  STRUCT
   HLINE_DX : STRUCT
    REP_SEL : BOOL ;
    S02_SEL : BOOL ;
    S03_SEL : BOOL ;
    RC2_SEL : BOOL ;
    BUF2_SEL : BOOL ;
    S04_SEL : BOOL ;
    S05_SEL : BOOL ;
    TT_SEL : BOOL ;
    SPARE : BOOL ;
    SPARE1 : BOOL ;
    SPARE2 : BOOL ;
    SPARE3 : BOOL ;
    SPARE4 : BOOL ;
    SPARE5 : BOOL ;
    SPARE6 : BOOL ;
    SPARE7 : BOOL ;
    SPARE8 : BOOL ;
    SPARE9 : BOOL ;
    SPARE10 : BOOL ;
    SPARE11 : BOOL ;
    SPARE12 : BOOL ;
    SPARE13 : BOOL ;
    SPARE14 : BOOL ;
    SPARE15 : BOOL ;
    SPARE16 : BOOL ;
    SPARE17 : BOOL ;
    SPARE18 : BOOL ;
    SPARE19 : BOOL ;
    SPARE20 : BOOL ;
    SPARE21 : BOOL ;
    PB_ADV : BOOL ;
    PB_RET : BOOL ;
    LCK1_SEL : BOOL ;
    STP1_SEL : BOOL ;
    LCK2_SEL : BOOL ;
    STP2_SEL : BOOL ;
    LCK3_SEL : BOOL ;
    STP3_SEL : BOOL ;
    LCK4_SEL : BOOL ;
    STP4_SEL : BOOL ;
    ELE_SEL : BOOL ;
    RC_SEL : BOOL ;
    HK_SEL : BOOL ;
    PLOCK_SEL : BOOL ;
    MOTOR_SEL : BOOL ;
    SPARE37 : BOOL ;
    SPARE38 : BOOL ;
    SPARE39 : BOOL ;
    SPARE40 : BOOL ;
    SPARE41 : BOOL ;
    SPARE42 : BOOL ;
    SPARE43 : BOOL ;
    SPARE44 : BOOL ;
    SPARE45 : BOOL ;
    SPARE46 : BOOL ;
    SPARE47 : BOOL ;
    SPARE48 : BOOL ;
    SPARE49 : BOOL ;
    SPARE50 : BOOL ;
    SPARE51 : BOOL ;
    SPARE52 : BOOL ;
    SPARE53 : BOOL ;
    SPARE54 : BOOL ;
    SPARE55 : BOOL ;
    REP_LCK1_SEL : BOOL ;
    REP_STP1_SEL : BOOL ;
    REP_LCK2_SEL : BOOL ;
    REP_STP2_SEL : BOOL ;
    SPARE60 : BOOL ;
    SPARE61 : BOOL ;
    SPARE62 : BOOL ;
    SPARE63 : BOOL ;
    REP_ELE_SEL : BOOL ;
    REP_RC_SEL : BOOL ;
    SPARE66 : BOOL ;
    SPARE67 : BOOL ;
    SPARE68 : BOOL ;
    SPARE69 : BOOL ;
    SPARE70 : BOOL ;
    SPARE71 : BOOL ;
    S02_LCK1_SEL : BOOL ;
    S02_STP1_SEL : BOOL ;
    S02_LCK2_SEL : BOOL ;
    S02_STP2_SEL : BOOL ;
    S02_LCK3_SEL : BOOL ;
    S02_STP3_SEL : BOOL ;
    SPARE78 : BOOL ;
    SPARE79 : BOOL ;
    S02_ELE_SEL : BOOL ;
    S02_RC_SEL : BOOL ;
    SPARE22 : BOOL ;
    SPARE23 : BOOL ;
    SPARE84 : BOOL ;
    SPARE85 : BOOL ;
    SPARE86 : BOOL ;
    SPARE87 : BOOL ;
    S03_LCK1_SEL : BOOL ;
    S03_STP1_SEL : BOOL ;
    SPARE90 : BOOL ;
    SPARE91 : BOOL ;
    SPARE92 : BOOL ;
    SPARE93 : BOOL ;
    SPARE94 : BOOL ;
    SPARE95 : BOOL ;
    S03_ELE_SEL : BOOL ;
    SPARE97 : BOOL ;
    SPARE98 : BOOL ;
    SPARE99 : BOOL ;
    SPARE100 : BOOL ;
    SPARE101 : BOOL ;
    SPARE102 : BOOL ;
    SPARE103 : BOOL ;
    RC2_LCK1_SEL : BOOL ;
    RC2_STP1_SEL : BOOL ;
    RC2_LCK2_SEL : BOOL ;
    RC2_STP2_SEL : BOOL ;
    RC2_LCK3_SEL : BOOL ;
    RC2_STP3_SEL : BOOL ;
    RC2_LCK4_SEL : BOOL ;
    RC2_STP4_SEL : BOOL ;
    SPARE112 : BOOL ;
    RC2_RC_SEL : BOOL ;
    SPARE114 : BOOL ;
    SPARE115 : BOOL ;
    SPARE116 : BOOL ;
    SPARE117 : BOOL ;
    SPARE118 : BOOL ;
    SPARE119 : BOOL ;
    BUF1_LCK1_SEL : BOOL ;
    BUF1_STP1_SEL : BOOL ;
    SPARE122 : BOOL ;
    SPARE123 : BOOL ;
    SPARE124 : BOOL ;
    SPARE125 : BOOL ;
    SPARE126 : BOOL ;
    SPARE127 : BOOL ;
    SPARE128 : BOOL ;
    SPARE129 : BOOL ;
    SPARE130 : BOOL ;
    SPARE131 : BOOL ;
    SPARE132 : BOOL ;
    SPARE133 : BOOL ;
    SPARE134 : BOOL ;
    SPARE135 : BOOL ;
    BUF2_LCK1_SEL : BOOL ;
    BUF2_STP1_SEL : BOOL ;
    SPARE138 : BOOL ;
    SPARE139 : BOOL ;
    SPARE140 : BOOL ;
    SPARE141 : BOOL ;
    SPARE142 : BOOL ;
    SPARE143 : BOOL ;
    SPARE144 : BOOL ;
    SPARE145 : BOOL ;
    SPARE146 : BOOL ;
    SPARE147 : BOOL ;
    SPARE148 : BOOL ;
    SPARE149 : BOOL ;
    SPARE150 : BOOL ;
    SPARE151 : BOOL ;
    S04_LCK1_SEL : BOOL ;
    S04_STP1_SEL : BOOL ;
    SPARE154 : BOOL ;
    SPARE155 : BOOL ;
    SPARE156 : BOOL ;
    SPARE157 : BOOL ;
    SPARE158 : BOOL ;
    SPARE159 : BOOL ;
    S04_ELE_SEL : BOOL ;
    SPARE161 : BOOL ;
    S04_HK_SEL : BOOL ;
    SPARE163 : BOOL ;
    SPARE164 : BOOL ;
    SPARE165 : BOOL ;
    SPARE166 : BOOL ;
    SPARE167 : BOOL ;
    S05_LCK1_SEL : BOOL ;
    S05_STP1_SEL : BOOL ;
    SPARE170 : BOOL ;
    SPARE171 : BOOL ;
    SPARE172 : BOOL ;
    SPARE173 : BOOL ;
    SPARE174 : BOOL ;
    SPARE175 : BOOL ;
    S05_ELE_SEL : BOOL ;
    SPARE177 : BOOL ;
    S05_HK_SEL : BOOL ;
    SPARE179 : BOOL ;
    SPARE180 : BOOL ;
    SPARE181 : BOOL ;
    SPARE182 : BOOL ;
    SPARE183 : BOOL ;
    TT_PLOCK_SEL : BOOL ;
    TT_ELE_SEL : BOOL ;
    TT_ROLL_SEL : BOOL ;
    SPARE187 : BOOL ;
    SPARE188 : BOOL ;
    SPARE189 : BOOL ;
    SPARE190 : BOOL ;
    SPARE191 : BOOL ;
    SPARE192 : BOOL ;
    SPARE193 : BOOL ;
    SPARE194 : BOOL ;
    SPARE195 : BOOL ;
    SPARE196 : BOOL ;
    SPARE197 : BOOL ;
    SPARE198 : BOOL ;
    SPARE199 : BOOL ;
    SPARE200 : BOOL ;
    SPARE201 : BOOL ;
    SPARE202 : BOOL ;
    SPARE203 : BOOL ;
    SPARE204 : BOOL ;
    SPARE205 : BOOL ;
    SPARE206 : BOOL ;
    SPARE207 : BOOL ;
    SPARE208 : BOOL ;
    SPARE209 : BOOL ;
    SPARE210 : BOOL ;
    SPARE211 : BOOL ;
    SPARE212 : BOOL ;
    SPARE213 : BOOL ;
    SPARE214 : BOOL ;
    SPARE215 : BOOL ;
    SPARE216 : BOOL ;
    SPARE217 : BOOL ;
    SPARE218 : BOOL ;
    SPARE219 : BOOL ;
    SPARE220 : BOOL ;
    SPARE221 : BOOL ;
    SPARE222 : BOOL ;
    SPARE223 : BOOL ;
    SPARE224 : BOOL ;
    SPARE225 : BOOL ;
    SPARE226 : BOOL ;
    SPARE227 : BOOL ;
    SPARE228 : BOOL ;
    SPARE229 : BOOL ;
    SPARE230 : BOOL ;
    SPARE231 : BOOL ;
    SPARE232 : BOOL ;
    SPARE233 : BOOL ;
    SPARE234 : BOOL ;
    SPARE235 : BOOL ;
    SPARE236 : BOOL ;
    SPARE237 : BOOL ;
    SPARE238 : BOOL ;
    SPARE239 : BOOL ;
    SPARE240 : BOOL ;
    SPARE241 : BOOL ;
    SPARE242 : BOOL ;
    SPARE243 : BOOL ;
    SPARE244 : BOOL ;
    SPARE245 : BOOL ;
    SPARE246 : BOOL ;
    SPARE247 : BOOL ;
    SPARE248 : BOOL ;
    SPARE249 : BOOL ;
    SPARE250 : BOOL ;
    SPARE251 : BOOL ;
    SPARE252 : BOOL ;
    SPARE253 : BOOL ;
    SPARE254 : BOOL ;
    SPARE255 : BOOL ;
    SPARE256 : BOOL ;
    SPARE257 : BOOL ;
    SPARE258 : BOOL ;
    SPARE259 : BOOL ;
    SPARE260 : BOOL ;
    SPARE261 : BOOL ;
    SPARE262 : BOOL ;
    SPARE263 : BOOL ;
    SPARE264 : BOOL ;
    SPARE265 : BOOL ;
    SPARE266 : BOOL ;
    SPARE267 : BOOL ;
    SPARE268 : BOOL ;
    SPARE269 : BOOL ;
    SPARE270 : BOOL ;
    SPARE271 : BOOL ;
    SPARE272 : BOOL ;
    SPARE273 : BOOL ;
    SPARE274 : BOOL ;
    SPARE275 : BOOL ;
    SPARE276 : BOOL ;
    SPARE277 : BOOL ;
    SPARE278 : BOOL ;
    SPARE279 : BOOL ;
    SPARE280 : BOOL ;
    SPARE281 : BOOL ;
    SPARE282 : BOOL ;
    SPARE283 : BOOL ;
    SPARE284 : BOOL ;
    SPARE285 : BOOL ;
    SPARE286 : BOOL ;
    SPARE287 : BOOL ;
    SPARE288 : BOOL ;
    SPARE289 : BOOL ;
    SPARE290 : BOOL ;
    SPARE291 : BOOL ;
    SPARE292 : BOOL ;
    SPARE293 : BOOL ;
    SPARE294 : BOOL ;
    SPARE295 : BOOL ;
    SPARE296 : BOOL ;
    SPARE297 : BOOL ;
    SPARE298 : BOOL ;
    SPARE299 : BOOL ;
    SPARE300 : BOOL ;
    SPARE301 : BOOL ;
    SPARE302 : BOOL ;
    SPARE303 : BOOL ;
    SPARE304 : BOOL ;
    SPARE305 : BOOL ;
    SPARE306 : BOOL ;
    SPARE307 : BOOL ;
    SPARE308 : BOOL ;
    SPARE309 : BOOL ;
    SPARE310 : BOOL ;
   END_STRUCT ;
   HLINE_DW : STRUCT
    REP_LCK1_A_LAMP : WORD ;
    REP_LCK1_R_LAMP : WORD ;
    REP_STP1_A_LAMP : WORD ;
    REP_STP1_R_LAMP : WORD ;
    REP_LCK2_A_LAMP : WORD ;
    REP_LCK2_R_LAMP : WORD ;
    REP_STP2_A_LAMP : WORD ;
    REP_STP2_R_LAMP : WORD ;
    REP_ELE_A_LAMP : WORD ;
    REP_ELE_R_LAMP : WORD ;
    REP_RC_A_LAMP : WORD ;
    REP_RC_R_LAMP : WORD ;
    SPARE_WORD1 : WORD ;
    SPARE_WORD2 : WORD ;
    SPARE_WORD3 : WORD ;
    SPARE_WORD4 : WORD ;
    S02_LCK1_A_LAMP : WORD ;
    S02_LCK1_R_LAMP : WORD ;
    S02_STP1_A_LAMP : WORD ;
    S02_STP1_R_LAMP : WORD ;
    S02_LCK2_A_LAMP : WORD ;
    S02_LCK2_R_LAMP : WORD ;
    S02_STP2_A_LAMP : WORD ;
    S02_STP2_R_LAMP : WORD ;
    S02_LCK3_A_LAMP : WORD ;
    S02_LCK3_R_LAMP : WORD ;
    S02_STP3_A_LAMP : WORD ;
    S02_STP3_R_LAMP : WORD ;
    S02_ELE_A_LAMP : WORD ;
    S02_ELE_R_LAMP : WORD ;
    S02_RC_A_LAMP : WORD ;
    S02_RC_R_LAMP : WORD ;
    SPARE_WORD15 : WORD ;
    SPARE_WORD16 : WORD ;
    SPARE_WORD17 : WORD ;
    SPARE_WORD18 : WORD ;
    S03_LCK1_A_LAMP : WORD ;
    S03_LCK1_R_LAMP : WORD ;
    S03_STP1_A_LAMP : WORD ;
    S03_STP1_R_LAMP : WORD ;
    S03_ELE_A_LAMP : WORD ;
    S03_ELE_R_LAMP : WORD ;
    SPARE_WORD25 : WORD ;
    SPARE_WORD26 : WORD ;
    SPARE_WORD27 : WORD ;
    SPARE_WORD28 : WORD ;
    RC2_LCK1_A_LAMP : WORD ;
    RC2_LCK1_R_LAMP : WORD ;
    RC2_STP1_A_LAMP : WORD ;
    RC2_STP1_R_LAMP : WORD ;
    RC2_LCK2_A_LAMP : WORD ;
    RC2_LCK2_R_LAMP : WORD ;
    RC2_STP2_A_LAMP : WORD ;
    RC2_STP2_R_LAMP : WORD ;
    RC2_LCK3_A_LAMP1 : WORD ;
    RC2_LCK3_R_LAMP1 : WORD ;
    RC2_STP3_A_LAMP1 : WORD ;
    RC2_STP3_R_LAMP1 : WORD ;
    RC2_LCK4_A_LAMP1 : WORD ;
    RC2_LCK4_R_LAMP1 : WORD ;
    RC2_STP4_A_LAMP1 : WORD ;
    RC2_STP4_R_LAMP1 : WORD ;
    RC2_RC_A_LAMP1 : WORD ;
    RC2_RC_R_LAMP1 : WORD ;
    SPARE_WORD34 : WORD ;
    SPARE_WORD35 : WORD ;
    SPARE_WORD36 : WORD ;
    SPARE_WORD37 : WORD ;
    BUF1_LCK1_A_LAMP : WORD ;
    BUF1_LCK1_R_LAMP : WORD ;
    BUF1_STP1_A_LAMP : WORD ;
    BUF1_STP1_R_LAMP : WORD ;
    SPARE_WORD42 : WORD ;
    SPARE_WORD43 : WORD ;
    SPARE_WORD44 : WORD ;
    SPARE_WORD45 : WORD ;
    BUF2_LCK1_A_LAMP : WORD ;
    BUF2_LCK1_R_LAMP : WORD ;
    BUF2_STP1_A_LAMP : WORD ;
    BUF2_STP1_R_LAMP : WORD ;
    SPARE_WORD50 : WORD ;
    SPARE_WORD51 : WORD ;
    SPARE_WORD52 : WORD ;
    SPARE_WORD53 : WORD ;
    S04_LCK1_A_LAMP : WORD ;
    S04_LCK1_R_LAMP : WORD ;
    S04_STP1_A_LAMP : WORD ;
    S04_STP2_R_LAMP : WORD ;
    S04_ELE_A_LAMP : WORD ;
    S04_ELE_R_LAMP : WORD ;
    S04_HK_A_LAMP : WORD ;
    S04_HK_R_LAMP : WORD ;
    SPARE_WORD55 : WORD ;
    SPARE_WORD56 : WORD ;
    SPARE_WORD57 : WORD ;
    SPARE_WORD58 : WORD ;
    S05_LCK1_A_LAMP : WORD ;
    S05_LCK1_R_LAMP : WORD ;
    S05_STP1_A_LAMP : WORD ;
    S05_STP2_R_LAMP : WORD ;
    S05_ELE_A_LAMP : WORD ;
    S05_ELE_R_LAMP : WORD ;
    S05_HK_A_LAMP : WORD ;
    S05_HK_R_LAMP : WORD ;
    SPARE_WORD60 : WORD ;
    SPARE_WORD61 : WORD ;
    SPARE_WORD62 : WORD ;
    SPARE_WORD63 : WORD ;
    TT_PLOCK_A_LAMP : WORD ;
    TT_PLOCK_R_LAMP : WORD ;
    TT_ELE_A_LAMP : WORD ;
    TT_ELE_R_LAMP : WORD ;
    TT_ROLL_A_LAMP : WORD ;
    TT_ROLL_R_LAMP : WORD ;
    SPARE_WORD70 : WORD ;
    SPARE_WORD71 : WORD ;
    SPARE_WORD72 : WORD ;
    SPARE_WORD73 : WORD ;
    SPARE_WORD74 : WORD ;
    SPARE_WORD75 : WORD ;
    SPARE_WORD76 : WORD ;
    SPARE_WORD77 : WORD ;
    SPARE_WORD78 : WORD ;
    SPARE_WORD79 : WORD ;
    SPARE_WORD80 : WORD ;
    SPARE_WORD81 : WORD ;
    SPARE_WORD82 : WORD ;
    SPARE_WORD83 : WORD ;
    SPARE_WORD84 : WORD ;
    SPARE_WORD85 : WORD ;
    SPARE_WORD86 : WORD ;
    SPARE_WORD87 : WORD ;
    SPARE_WORD88 : WORD ;
    SPARE_WORD89 : WORD ;
    SPARE_WORD90 : WORD ;
    SPARE_WORD91 : WORD ;
    SPARE_WORD92 : WORD ;
    SPARE_WORD93 : WORD ;
    SPARE_WORD94 : WORD ;
    SPARE_WORD95 : WORD ;
    SPARE_WORD96 : WORD ;
    SPARE_WORD97 : WORD ;
    SPARE_WORD98 : WORD ;
    SPARE_WORD99 : WORD ;
    SPARE_WORD100 : WORD ;
    SPARE_WORD101 : WORD ;
    SPARE_WORD102 : WORD ;
    SPARE_WORD103 : WORD ;
    SPARE_WORD104 : WORD ;
    SPARE_WORD105 : WORD ;
    SPARE_WORD106 : WORD ;
    SPARE_WORD107 : WORD ;
    SPARE_WORD108 : WORD ;
    SPARE_WORD109 : WORD ;
    SPARE_WORD110 : WORD ;
    SPARE_WORD111 : WORD ;
    SPARE_WORD112 : WORD ;
    SPARE_WORD113 : WORD ;
    SPARE_WORD114 : WORD ;
    SPARE_WORD115 : WORD ;
    SPARE_WORD116 : WORD ;
    SPARE_WORD117 : WORD ;
    SPARE_WORD118 : WORD ;
    SPARE_WORD119 : WORD ;
    SPARE_WORD120 : WORD ;
    SPARE_WORD121 : WORD ;
    SPARE_WORD122 : WORD ;
    SPARE_WORD123 : WORD ;
    SPARE_WORD124 : WORD ;
    SPARE_WORD125 : WORD ;
    SPARE_WORD126 : WORD ;
    SPARE_WORD127 : WORD ;
    SPARE_WORD128 : WORD ;
    SPARE_WORD129 : WORD ;
    SPARE_WORD130 : WORD ;
    SPARE_WORD131 : WORD ;
    SPARE_WORD132 : WORD ;
    SPARE_WORD133 : WORD ;
    SPARE_WORD134 : WORD ;
    SPARE_WORD135 : WORD ;
   END_STRUCT ;
   HUPDL_DX : STRUCT
    _1ST_U_SEL : BOOL ;
    _2ND_U1_SEL : BOOL ;
    _2ND_U2_SEL : BOOL ;
    SPUSH1_SEL : BOOL ;
    LOCKG_SEL : BOOL ;
    SPARE1 : BOOL ;
    SPARE2 : BOOL ;
    SPARE3 : BOOL ;
    Q_1ST_PIN_SEL : BOOL ;
    Q_2ND_UNIT_SEL : BOOL ;
    Q_3RD_UNIT_SEL : BOOL ;
    Q_4TH_UNIT_SEL : BOOL ;
    SPARE8 : BOOL ;
    SPARE9 : BOOL ;
    SPARE10 : BOOL ;
    SPARE11 : BOOL ;
    SPARE12 : BOOL ;
    SPARE13 : BOOL ;
    SPARE14 : BOOL ;
    SPARE15 : BOOL ;
    SPARE16 : BOOL ;
    SPARE17 : BOOL ;
    SPARE18 : BOOL ;
    SPARE19 : BOOL ;
    SPARE20 : BOOL ;
    SPARE21 : BOOL ;
    SPARE22 : BOOL ;
    SPARE23 : BOOL ;
    SPARE24 : BOOL ;
    SPARE25 : BOOL ;
    PB_ADV : BOOL ;
    PB_RET : BOOL ;
    BH_1_SEL : BOOL ;
    BH_2_SEL : BOOL ;
    BH_3_SEL : BOOL ;
    BH_4_SEL : BOOL ;
    BH_5_SEL : BOOL ;
    BH_6_SEL : BOOL ;
    BH_7_SEL : BOOL ;
    BH_8_SEL : BOOL ;
    BH_9_SEL : BOOL ;
    BH_10_SEL : BOOL ;
    BH_11_SEL : BOOL ;
    BH_12_SEL : BOOL ;
    BH_13_SEL : BOOL ;
    BH_14_SEL : BOOL ;
    BH_15_SEL : BOOL ;
    BH_16_SEL : BOOL ;
    SPARE42 : BOOL ;
    SPARE43 : BOOL ;
    SPARE44 : BOOL ;
    SPARE45 : BOOL ;
    SPARE46 : BOOL ;
    SPARE47 : BOOL ;
    SPARE48 : BOOL ;
    SPARE49 : BOOL ;
    SPARE50 : BOOL ;
    SPARE51 : BOOL ;
    SPARE52 : BOOL ;
    SPARE53 : BOOL ;
    SPARE54 : BOOL ;
    SPARE55 : BOOL ;
    SPARE56 : BOOL ;
    SPARE57 : BOOL ;
    VI_1_SEL : BOOL ;
    VI_2_SEL : BOOL ;
    VI_3_SEL : BOOL ;
    VI_4_SEL : BOOL ;
    VI_5_SEL : BOOL ;
    VI_6_SEL : BOOL ;
    VI_7_SEL : BOOL ;
    VI_8_SEL : BOOL ;
    VI_9_SEL : BOOL ;
    VI_10_SEL : BOOL ;
    VI_11_SEL : BOOL ;
    VI_12_SEL : BOOL ;
    VI_13_SEL : BOOL ;
    VI_14_SEL : BOOL ;
    VI_15_SEL : BOOL ;
    VI_16_SEL : BOOL ;
    SPARE59 : BOOL ;
    SPARE60 : BOOL ;
    SPARE61 : BOOL ;
    SPARE62 : BOOL ;
    SPARE63 : BOOL ;
    SPARE64 : BOOL ;
    SPARE65 : BOOL ;
    SPARE66 : BOOL ;
    SPARE67 : BOOL ;
    SPARE68 : BOOL ;
    SPARE69 : BOOL ;
    SPARE70 : BOOL ;
    SPARE71 : BOOL ;
    SPARE72 : BOOL ;
    SPARE73 : BOOL ;
    SPARE74 : BOOL ;
    SPARE75 : BOOL ;
    SPARE76 : BOOL ;
    SPARE77 : BOOL ;
    SPARE78 : BOOL ;
    SPARE79 : BOOL ;
    SPARE80 : BOOL ;
    SPARE81 : BOOL ;
    SPARE82 : BOOL ;
    SPARE83 : BOOL ;
    SPARE84 : BOOL ;
    SPARE85 : BOOL ;
    SPARE86 : BOOL ;
    SPARE87 : BOOL ;
    SPARE88 : BOOL ;
    SPARE89 : BOOL ;
    SPARE90 : BOOL ;
    SPARE91 : BOOL ;
    SPARE92 : BOOL ;
    SPARE93 : BOOL ;
    SPARE94 : BOOL ;
    SPARE95 : BOOL ;
    SPARE96 : BOOL ;
    SPARE97 : BOOL ;
    SPARE98 : BOOL ;
    SPARE99 : BOOL ;
    SPARE100 : BOOL ;
    SPARE101 : BOOL ;
    SPARE102 : BOOL ;
    SPARE103 : BOOL ;
    SPARE104 : BOOL ;
    SPARE105 : BOOL ;
    SPARE106 : BOOL ;
    SPARE107 : BOOL ;
    SPARE108 : BOOL ;
    SPARE109 : BOOL ;
    SPARE110 : BOOL ;
    SPARE111 : BOOL ;
    SPARE112 : BOOL ;
    SPARE113 : BOOL ;
    SPARE114 : BOOL ;
    SPARE115 : BOOL ;
    SPARE116 : BOOL ;
    SPARE117 : BOOL ;
    SPARE118 : BOOL ;
    SPARE119 : BOOL ;
    SPARE120 : BOOL ;
    SPARE121 : BOOL ;
    SPARE122 : BOOL ;
    SPARE123 : BOOL ;
    SPARE124 : BOOL ;
    SPARE125 : BOOL ;
    SPARE126 : BOOL ;
    SPARE127 : BOOL ;
    SPARE128 : BOOL ;
    SPARE129 : BOOL ;
    SPARE130 : BOOL ;
    SPARE131 : BOOL ;
    SPARE132 : BOOL ;
    SPARE133 : BOOL ;
    SPARE134 : BOOL ;
    SPARE135 : BOOL ;
    SPARE136 : BOOL ;
    SPARE137 : BOOL ;
    SPARE138 : BOOL ;
   END_STRUCT ;
   HUPDL_DW : STRUCT
    _1ST_U_ADV_LAMP : WORD ;
    _1ST_U_RET_LAMP : WORD ;
    _2ND_U1_ADV_LAMP : WORD ;
    _2ND_U1_RET_LAMP : WORD ;
    _2ND_U2_ADV_LAMP : WORD ;
    _2ND_U2_RET_LAMP : WORD ;
    SPUSH1_ADV_LAMP : WORD ;
    SPUSH1_RET_LAMP : WORD ;
    LOCKG_ADV_LAMP : WORD ;
    LOCKG_RET_LAMP : WORD ;
    SPARE_WORD2 : WORD ;
    SPARE_WORD3 : WORD ;
    SPARE_WORD4 : WORD ;
    SPARE_WORD5 : WORD ;
    SPARE_WORD6 : WORD ;
    SPARE_WORD7 : WORD ;
    SPARE_WORD8 : WORD ;
    SPARE_WORD9 : WORD ;
    SPARE_WORD10 : WORD ;
    SPARE_WORD11 : WORD ;
    Q_1ST_PIN_ADV_LAMP : WORD ;
    Q_1ST_PIN_RET_LAMP : WORD ;
    Q_2ND_UNIT_ADV_LAMP : WORD ;
    Q_2ND_UNIT_RET_LAMP : WORD ;
    Q_3RD_UNIT_ADV_LAMP : WORD ;
    Q_3RD_UNIT_RET_LAMP : WORD ;
    Q_4TH_UNIT_ADV_LAMP : WORD ;
    Q_4TH_UNIT_RET_LAMP : WORD ;
    SPARE_WORD20 : WORD ;
    SPARE_WORD21 : WORD ;
    SPARE_WORD22 : WORD ;
    SPARE_WORD23 : WORD ;
    BH_1_ADV_LAMP : WORD ;
    BH_1_RET_LAMP : WORD ;
    BH_2_ADV_LAMP : WORD ;
    BH_2_RET_LAMP : WORD ;
    BH_3_ADV_LAMP : WORD ;
    BH_3_RET_LAMP : WORD ;
    BH_4_ADV_LAMP : WORD ;
    BH_4_RET_LAMP : WORD ;
    BH_5_ADV_LAMP : WORD ;
    BH_5_RET_LAMP : WORD ;
    BH_6_ADV_LAMP : WORD ;
    BH_6_RET_LAMP : WORD ;
    BH_7_ADV_LAMP : WORD ;
    BH_7_RET_LAMP : WORD ;
    BH_8_ADV_LAMP : WORD ;
    BH_8_RET_LAMP : WORD ;
    BH_9_ADV_LAMP : WORD ;
    BH_9_RET_LAMP : WORD ;
    BH_10_ADV_LAMP : WORD ;
    BH_10_RET_LAMP : WORD ;
    SPARE_WORD54 : WORD ;
    SPARE_WORD55 : WORD ;
    SPARE_WORD56 : WORD ;
    SPARE_WORD57 : WORD ;
    SPARE_WORD58 : WORD ;
    SPARE_WORD59 : WORD ;
    SPARE_WORD60 : WORD ;
    SPARE_WORD61 : WORD ;
    SPARE_WORD62 : WORD ;
    SPARE_WORD63 : WORD ;
    SPARE_WORD64 : WORD ;
    SPARE_WORD65 : WORD ;
    SPARE_WORD66 : WORD ;
    SPARE_WORD67 : WORD ;
    SPARE_WORD68 : WORD ;
    SPARE_WORD69 : WORD ;
    SPARE_WORD70 : WORD ;
    SPARE_WORD71 : WORD ;
    SPARE_WORD72 : WORD ;
    SPARE_WORD73 : WORD ;
    SPARE_WORD74 : WORD ;
    SPARE_WORD75 : WORD ;
    SPARE_WORD76 : WORD ;
    SPARE_WORD77 : WORD ;
    SPARE_WORD78 : WORD ;
    SPARE_WORD79 : WORD ;
    SPARE_WORD80 : WORD ;
    SPARE_WORD81 : WORD ;
    SPARE_WORD82 : WORD ;
    SPARE_WORD83 : WORD ;
    SPARE_WORD84 : WORD ;
    SPARE_WORD85 : WORD ;
    SPARE_WORD86 : WORD ;
    SPARE_WORD87 : WORD ;
    SPARE_WORD88 : WORD ;
    SPARE_WORD89 : WORD ;
    SPARE_WORD90 : WORD ;
    SPARE_WORD91 : WORD ;
    SPARE_WORD92 : WORD ;
    SPARE_WORD93 : WORD ;
    SPARE_WORD94 : WORD ;
    SPARE_WORD95 : WORD ;
    SPARE_WORD96 : WORD ;
    SPARE_WORD97 : WORD ;
    SPARE_WORD98 : WORD ;
    SPARE_WORD99 : WORD ;
    SPARE_WORD100 : WORD ;
    SPARE_WORD101 : WORD ;
    SPARE_WORD102 : WORD ;
    SPARE_WORD103 : WORD ;
    SPARE_WORD104 : WORD ;
    SPARE_WORD105 : WORD ;
    SPARE_WORD106 : WORD ;
    SPARE_WORD107 : WORD ;
    SPARE_WORD108 : WORD ;
    SPARE_WORD109 : WORD ;
    SPARE_WORD110 : WORD ;
    SPARE_WORD111 : WORD ;
    SPARE_WORD112 : WORD ;
    SPARE_WORD113 : WORD ;
    SPARE_WORD114 : WORD ;
    SPARE_WORD115 : WORD ;
    SPARE_WORD116 : WORD ;
    SPARE_WORD117 : WORD ;
    SPARE_WORD118 : WORD ;
    SPARE_WORD119 : WORD ;
    SPARE_WORD120 : WORD ;
    SPARE_WORD121 : WORD ;
    SPARE_WORD122 : WORD ;
    SPARE_WORD123 : WORD ;
    SPARE_WORD124 : WORD ;
    SPARE_WORD125 : WORD ;
    SPARE_WORD126 : WORD ;
    SPARE_WORD127 : WORD ;
    SPARE_WORD128 : WORD ;
    SPARE_WORD129 : WORD ;
    SPARE_WORD130 : WORD ;
    SPARE_WORD131 : WORD ;
    SPARE_WORD132 : WORD ;
    SPARE_WORD133 : WORD ;
    SPARE_WORD134 : WORD ;
    SPARE_WORD135 : WORD ;
    SPARE_WORD136 : WORD ;
    SPARE_WORD137 : WORD ;
    SPARE_WORD138 : WORD ;
    SPARE_WORD139 : WORD ;
    SPARE_WORD140 : WORD ;
    SPARE_WORD141 : WORD ;
    SPARE_WORD142 : WORD ;
    SPARE_WORD143 : WORD ;
    SPARE_WORD144 : WORD ;
    SPARE_WORD145 : WORD ;
    SPARE_WORD146 : WORD ;
    SPARE_WORD147 : WORD ;
    SPARE_WORD148 : WORD ;
    SPARE_WORD149 : WORD ;
    SPARE_WORD150 : WORD ;
    SPARE_WORD151 : WORD ;
    SPARE_WORD152 : WORD ;
    SPARE_WORD153 : WORD ;
    SPARE_WORD154 : WORD ;
    SPARE_WORD155 : WORD ;
    SPARE_WORD156 : WORD ;
    SPARE_WORD157 : WORD ;
    SPARE_WORD158 : WORD ;
    SPARE_WORD159 : WORD ;
    SPARE_WORD160 : WORD ;
    SPARE_WORD161 : WORD ;
    SPARE_WORD162 : WORD ;
    SPARE_WORD163 : WORD ;
    SPARE_WORD164 : WORD ;
    SPARE_WORD165 : WORD ;
    SPARE_WORD166 : WORD ;
    SPARE_WORD167 : WORD ;
    SPARE_WORD168 : WORD ;
    SPARE_WORD169 : WORD ;
    SPARE_WORD170 : WORD ;
    SPARE_WORD171 : WORD ;
    SPARE_WORD172 : WORD ;
    SPARE_WORD173 : WORD ;
    SPARE_WORD174 : WORD ;
    SPARE_WORD175 : WORD ;
    SPARE_WORD176 : WORD ;
    SPARE_WORD177 : WORD ;
    SPARE_WORD178 : WORD ;
    SPARE_WORD179 : WORD ;
    SPARE_WORD180 : WORD ;
    SPARE_WORD181 : WORD ;
   END_STRUCT ;
  END_STRUCT ;
BEGIN
   HLINE_DX.REP_SEL := FALSE;
   HLINE_DX.S02_SEL := FALSE;
   HLINE_DX.S03_SEL := FALSE;
   HLINE_DX.RC2_SEL := FALSE;
   HLINE_DX.BUF2_SEL := FALSE;
   HLINE_DX.S04_SEL := FALSE;
   HLINE_DX.S05_SEL := FALSE;
   HLINE_DX.TT_SEL := FALSE;
   HLINE_DX.SPARE := FALSE;
   HLINE_DX.SPARE1 := FALSE;
   HLINE_DX.SPARE2 := FALSE;
   HLINE_DX.SPARE3 := FALSE;
   HLINE_DX.SPARE4 := FALSE;
   HLINE_DX.SPARE5 := FALSE;
   HLINE_DX.SPARE6 := FALSE;
   HLINE_DX.SPARE7 := FALSE;
   HLINE_DX.SPARE8 := FALSE;
   HLINE_DX.SPARE9 := FALSE;
   HLINE_DX.SPARE10 := FALSE;
   HLINE_DX.SPARE11 := FALSE;
   HLINE_DX.SPARE12 := FALSE;
   HLINE_DX.SPARE13 := FALSE;
   HLINE_DX.SPARE14 := FALSE;
   HLINE_DX.SPARE15 := FALSE;
   HLINE_DX.SPARE16 := FALSE;
   HLINE_DX.SPARE17 := FALSE;
   HLINE_DX.SPARE18 := FALSE;
   HLINE_DX.SPARE19 := FALSE;
   HLINE_DX.SPARE20 := FALSE;
   HLINE_DX.SPARE21 := FALSE;
   HLINE_DX.PB_ADV := FALSE;
   HLINE_DX.PB_RET := FALSE;
   HLINE_DX.LCK1_SEL := FALSE;
   HLINE_DX.STP1_SEL := FALSE;
   HLINE_DX.LCK2_SEL := FALSE;
   HLINE_DX.STP2_SEL := FALSE;
   HLINE_DX.LCK3_SEL := FALSE;
   HLINE_DX.STP3_SEL := FALSE;
   HLINE_DX.LCK4_SEL := FALSE;
   HLINE_DX.STP4_SEL := FALSE;
   HLINE_DX.ELE_SEL := FALSE;
   HLINE_DX.RC_SEL := FALSE;
   HLINE_DX.HK_SEL := FALSE;
   HLINE_DX.PLOCK_SEL := FALSE;
   HLINE_DX.MOTOR_SEL := FALSE;
   HLINE_DX.SPARE37 := FALSE;
   HLINE_DX.SPARE38 := FALSE;
   HLINE_DX.SPARE39 := FALSE;
   HLINE_DX.SPARE40 := FALSE;
   HLINE_DX.SPARE41 := FALSE;
   HLINE_DX.SPARE42 := FALSE;
   HLINE_DX.SPARE43 := FALSE;
   HLINE_DX.SPARE44 := FALSE;
   HLINE_DX.SPARE45 := FALSE;
   HLINE_DX.SPARE46 := FALSE;
   HLINE_DX.SPARE47 := FALSE;
   HLINE_DX.SPARE48 := FALSE;
   HLINE_DX.SPARE49 := FALSE;
   HLINE_DX.SPARE50 := FALSE;
   HLINE_DX.SPARE51 := FALSE;
   HLINE_DX.SPARE52 := FALSE;
   HLINE_DX.SPARE53 := FALSE;
   HLINE_DX.SPARE54 := FALSE;
   HLINE_DX.SPARE55 := FALSE;
   HLINE_DX.REP_LCK1_SEL := FALSE;
   HLINE_DX.REP_STP1_SEL := FALSE;
   HLINE_DX.REP_LCK2_SEL := FALSE;
   HLINE_DX.REP_STP2_SEL := FALSE;
   HLINE_DX.SPARE60 := FALSE;
   HLINE_DX.SPARE61 := FALSE;
   HLINE_DX.SPARE62 := FALSE;
   HLINE_DX.SPARE63 := FALSE;
   HLINE_DX.REP_ELE_SEL := FALSE;
   HLINE_DX.REP_RC_SEL := FALSE;
   HLINE_DX.SPARE66 := FALSE;
   HLINE_DX.SPARE67 := FALSE;
   HLINE_DX.SPARE68 := FALSE;
   HLINE_DX.SPARE69 := FALSE;
   HLINE_DX.SPARE70 := FALSE;
   HLINE_DX.SPARE71 := FALSE;
   HLINE_DX.S02_LCK1_SEL := FALSE;
   HLINE_DX.S02_STP1_SEL := FALSE;
   HLINE_DX.S02_LCK2_SEL := FALSE;
   HLINE_DX.S02_STP2_SEL := FALSE;
   HLINE_DX.S02_LCK3_SEL := FALSE;
   HLINE_DX.S02_STP3_SEL := FALSE;
   HLINE_DX.SPARE78 := FALSE;
   HLINE_DX.SPARE79 := FALSE;
   HLINE_DX.S02_ELE_SEL := FALSE;
   HLINE_DX.S02_RC_SEL := FALSE;
   HLINE_DX.SPARE22 := FALSE;
   HLINE_DX.SPARE23 := FALSE;
   HLINE_DX.SPARE84 := FALSE;
   HLINE_DX.SPARE85 := FALSE;
   HLINE_DX.SPARE86 := FALSE;
   HLINE_DX.SPARE87 := FALSE;
   HLINE_DX.S03_LCK1_SEL := FALSE;
   HLINE_DX.S03_STP1_SEL := FALSE;
   HLINE_DX.SPARE90 := FALSE;
   HLINE_DX.SPARE91 := FALSE;
   HLINE_DX.SPARE92 := FALSE;
   HLINE_DX.SPARE93 := FALSE;
   HLINE_DX.SPARE94 := FALSE;
   HLINE_DX.SPARE95 := FALSE;
   HLINE_DX.S03_ELE_SEL := FALSE;
   HLINE_DX.SPARE97 := FALSE;
   HLINE_DX.SPARE98 := FALSE;
   HLINE_DX.SPARE99 := FALSE;
   HLINE_DX.SPARE100 := FALSE;
   HLINE_DX.SPARE101 := FALSE;
   HLINE_DX.SPARE102 := FALSE;
   HLINE_DX.SPARE103 := FALSE;
   HLINE_DX.RC2_LCK1_SEL := FALSE;
   HLINE_DX.RC2_STP1_SEL := FALSE;
   HLINE_DX.RC2_LCK2_SEL := FALSE;
   HLINE_DX.RC2_STP2_SEL := FALSE;
   HLINE_DX.RC2_LCK3_SEL := FALSE;
   HLINE_DX.RC2_STP3_SEL := FALSE;
   HLINE_DX.RC2_LCK4_SEL := FALSE;
   HLINE_DX.RC2_STP4_SEL := FALSE;
   HLINE_DX.SPARE112 := FALSE;
   HLINE_DX.RC2_RC_SEL := FALSE;
   HLINE_DX.SPARE114 := FALSE;
   HLINE_DX.SPARE115 := FALSE;
   HLINE_DX.SPARE116 := FALSE;
   HLINE_DX.SPARE117 := FALSE;
   HLINE_DX.SPARE118 := FALSE;
   HLINE_DX.SPARE119 := FALSE;
   HLINE_DX.BUF1_LCK1_SEL := FALSE;
   HLINE_DX.BUF1_STP1_SEL := FALSE;
   HLINE_DX.SPARE122 := FALSE;
   HLINE_DX.SPARE123 := FALSE;
   HLINE_DX.SPARE124 := FALSE;
   HLINE_DX.SPARE125 := FALSE;
   HLINE_DX.SPARE126 := FALSE;
   HLINE_DX.SPARE127 := FALSE;
   HLINE_DX.SPARE128 := FALSE;
   HLINE_DX.SPARE129 := FALSE;
   HLINE_DX.SPARE130 := FALSE;
   HLINE_DX.SPARE131 := FALSE;
   HLINE_DX.SPARE132 := FALSE;
   HLINE_DX.SPARE133 := FALSE;
   HLINE_DX.SPARE134 := FALSE;
   HLINE_DX.SPARE135 := FALSE;
   HLINE_DX.BUF2_LCK1_SEL := FALSE;
   HLINE_DX.BUF2_STP1_SEL := FALSE;
   HLINE_DX.SPARE138 := FALSE;
   HLINE_DX.SPARE139 := FALSE;
   HLINE_DX.SPARE140 := FALSE;
   HLINE_DX.SPARE141 := FALSE;
   HLINE_DX.SPARE142 := FALSE;
   HLINE_DX.SPARE143 := FALSE;
   HLINE_DX.SPARE144 := FALSE;
   HLINE_DX.SPARE145 := FALSE;
   HLINE_DX.SPARE146 := FALSE;
   HLINE_DX.SPARE147 := FALSE;
   HLINE_DX.SPARE148 := FALSE;
   HLINE_DX.SPARE149 := FALSE;
   HLINE_DX.SPARE150 := FALSE;
   HLINE_DX.SPARE151 := FALSE;
   HLINE_DX.S04_LCK1_SEL := FALSE;
   HLINE_DX.S04_STP1_SEL := FALSE;
   HLINE_DX.SPARE154 := FALSE;
   HLINE_DX.SPARE155 := FALSE;
   HLINE_DX.SPARE156 := FALSE;
   HLINE_DX.SPARE157 := FALSE;
   HLINE_DX.SPARE158 := FALSE;
   HLINE_DX.SPARE159 := FALSE;
   HLINE_DX.S04_ELE_SEL := FALSE;
   HLINE_DX.SPARE161 := FALSE;
   HLINE_DX.S04_HK_SEL := FALSE;
   HLINE_DX.SPARE163 := FALSE;
   HLINE_DX.SPARE164 := FALSE;
   HLINE_DX.SPARE165 := FALSE;
   HLINE_DX.SPARE166 := FALSE;
   HLINE_DX.SPARE167 := FALSE;
   HLINE_DX.S05_LCK1_SEL := FALSE;
   HLINE_DX.S05_STP1_SEL := FALSE;
   HLINE_DX.SPARE170 := FALSE;
   HLINE_DX.SPARE171 := FALSE;
   HLINE_DX.SPARE172 := FALSE;
   HLINE_DX.SPARE173 := FALSE;
   HLINE_DX.SPARE174 := FALSE;
   HLINE_DX.SPARE175 := FALSE;
   HLINE_DX.S05_ELE_SEL := FALSE;
   HLINE_DX.SPARE177 := FALSE;
   HLINE_DX.S05_HK_SEL := FALSE;
   HLINE_DX.SPARE179 := FALSE;
   HLINE_DX.SPARE180 := FALSE;
   HLINE_DX.SPARE181 := FALSE;
   HLINE_DX.SPARE182 := FALSE;
   HLINE_DX.SPARE183 := FALSE;
   HLINE_DX.TT_PLOCK_SEL := FALSE;
   HLINE_DX.TT_ELE_SEL := FALSE;
   HLINE_DX.TT_ROLL_SEL := FALSE;
   HLINE_DX.SPARE187 := FALSE;
   HLINE_DX.SPARE188 := FALSE;
   HLINE_DX.SPARE189 := FALSE;
   HLINE_DX.SPARE190 := FALSE;
   HLINE_DX.SPARE191 := FALSE;
   HLINE_DX.SPARE192 := FALSE;
   HLINE_DX.SPARE193 := FALSE;
   HLINE_DX.SPARE194 := FALSE;
   HLINE_DX.SPARE195 := FALSE;
   HLINE_DX.SPARE196 := FALSE;
   HLINE_DX.SPARE197 := FALSE;
   HLINE_DX.SPARE198 := FALSE;
   HLINE_DX.SPARE199 := FALSE;
   HLINE_DX.SPARE200 := FALSE;
   HLINE_DX.SPARE201 := FALSE;
   HLINE_DX.SPARE202 := FALSE;
   HLINE_DX.SPARE203 := FALSE;
   HLINE_DX.SPARE204 := FALSE;
   HLINE_DX.SPARE205 := FALSE;
   HLINE_DX.SPARE206 := FALSE;
   HLINE_DX.SPARE207 := FALSE;
   HLINE_DX.SPARE208 := FALSE;
   HLINE_DX.SPARE209 := FALSE;
   HLINE_DX.SPARE210 := FALSE;
   HLINE_DX.SPARE211 := FALSE;
   HLINE_DX.SPARE212 := FALSE;
   HLINE_DX.SPARE213 := FALSE;
   HLINE_DX.SPARE214 := FALSE;
   HLINE_DX.SPARE215 := FALSE;
   HLINE_DX.SPARE216 := FALSE;
   HLINE_DX.SPARE217 := FALSE;
   HLINE_DX.SPARE218 := FALSE;
   HLINE_DX.SPARE219 := FALSE;
   HLINE_DX.SPARE220 := FALSE;
   HLINE_DX.SPARE221 := FALSE;
   HLINE_DX.SPARE222 := FALSE;
   HLINE_DX.SPARE223 := FALSE;
   HLINE_DX.SPARE224 := FALSE;
   HLINE_DX.SPARE225 := FALSE;
   HLINE_DX.SPARE226 := FALSE;
   HLINE_DX.SPARE227 := FALSE;
   HLINE_DX.SPARE228 := FALSE;
   HLINE_DX.SPARE229 := FALSE;
   HLINE_DX.SPARE230 := FALSE;
   HLINE_DX.SPARE231 := FALSE;
   HLINE_DX.SPARE232 := FALSE;
   HLINE_DX.SPARE233 := FALSE;
   HLINE_DX.SPARE234 := FALSE;
   HLINE_DX.SPARE235 := FALSE;
   HLINE_DX.SPARE236 := FALSE;
   HLINE_DX.SPARE237 := FALSE;
   HLINE_DX.SPARE238 := FALSE;
   HLINE_DX.SPARE239 := FALSE;
   HLINE_DX.SPARE240 := FALSE;
   HLINE_DX.SPARE241 := FALSE;
   HLINE_DX.SPARE242 := FALSE;
   HLINE_DX.SPARE243 := FALSE;
   HLINE_DX.SPARE244 := FALSE;
   HLINE_DX.SPARE245 := FALSE;
   HLINE_DX.SPARE246 := FALSE;
   HLINE_DX.SPARE247 := FALSE;
   HLINE_DX.SPARE248 := FALSE;
   HLINE_DX.SPARE249 := FALSE;
   HLINE_DX.SPARE250 := FALSE;
   HLINE_DX.SPARE251 := FALSE;
   HLINE_DX.SPARE252 := FALSE;
   HLINE_DX.SPARE253 := FALSE;
   HLINE_DX.SPARE254 := FALSE;
   HLINE_DX.SPARE255 := FALSE;
   HLINE_DX.SPARE256 := FALSE;
   HLINE_DX.SPARE257 := FALSE;
   HLINE_DX.SPARE258 := FALSE;
   HLINE_DX.SPARE259 := FALSE;
   HLINE_DX.SPARE260 := FALSE;
   HLINE_DX.SPARE261 := FALSE;
   HLINE_DX.SPARE262 := FALSE;
   HLINE_DX.SPARE263 := FALSE;
   HLINE_DX.SPARE264 := FALSE;
   HLINE_DX.SPARE265 := FALSE;
   HLINE_DX.SPARE266 := FALSE;
   HLINE_DX.SPARE267 := FALSE;
   HLINE_DX.SPARE268 := FALSE;
   HLINE_DX.SPARE269 := FALSE;
   HLINE_DX.SPARE270 := FALSE;
   HLINE_DX.SPARE271 := FALSE;
   HLINE_DX.SPARE272 := FALSE;
   HLINE_DX.SPARE273 := FALSE;
   HLINE_DX.SPARE274 := FALSE;
   HLINE_DX.SPARE275 := FALSE;
   HLINE_DX.SPARE276 := FALSE;
   HLINE_DX.SPARE277 := FALSE;
   HLINE_DX.SPARE278 := FALSE;
   HLINE_DX.SPARE279 := FALSE;
   HLINE_DX.SPARE280 := FALSE;
   HLINE_DX.SPARE281 := FALSE;
   HLINE_DX.SPARE282 := FALSE;
   HLINE_DX.SPARE283 := FALSE;
   HLINE_DX.SPARE284 := FALSE;
   HLINE_DX.SPARE285 := FALSE;
   HLINE_DX.SPARE286 := FALSE;
   HLINE_DX.SPARE287 := FALSE;
   HLINE_DX.SPARE288 := FALSE;
   HLINE_DX.SPARE289 := FALSE;
   HLINE_DX.SPARE290 := FALSE;
   HLINE_DX.SPARE291 := FALSE;
   HLINE_DX.SPARE292 := FALSE;
   HLINE_DX.SPARE293 := FALSE;
   HLINE_DX.SPARE294 := FALSE;
   HLINE_DX.SPARE295 := FALSE;
   HLINE_DX.SPARE296 := FALSE;
   HLINE_DX.SPARE297 := FALSE;
   HLINE_DX.SPARE298 := FALSE;
   HLINE_DX.SPARE299 := FALSE;
   HLINE_DX.SPARE300 := FALSE;
   HLINE_DX.SPARE301 := FALSE;
   HLINE_DX.SPARE302 := FALSE;
   HLINE_DX.SPARE303 := FALSE;
   HLINE_DX.SPARE304 := FALSE;
   HLINE_DX.SPARE305 := FALSE;
   HLINE_DX.SPARE306 := FALSE;
   HLINE_DX.SPARE307 := FALSE;
   HLINE_DX.SPARE308 := FALSE;
   HLINE_DX.SPARE309 := FALSE;
   HLINE_DX.SPARE310 := FALSE;
   HLINE_DW.REP_LCK1_A_LAMP := W#16#0;
   HLINE_DW.REP_LCK1_R_LAMP := W#16#0;
   HLINE_DW.REP_STP1_A_LAMP := W#16#0;
   HLINE_DW.REP_STP1_R_LAMP := W#16#0;
   HLINE_DW.REP_LCK2_A_LAMP := W#16#0;
   HLINE_DW.REP_LCK2_R_LAMP := W#16#0;
   HLINE_DW.REP_STP2_A_LAMP := W#16#0;
   HLINE_DW.REP_STP2_R_LAMP := W#16#0;
   HLINE_DW.REP_ELE_A_LAMP := W#16#0;
   HLINE_DW.REP_ELE_R_LAMP := W#16#0;
   HLINE_DW.REP_RC_A_LAMP := W#16#0;
   HLINE_DW.REP_RC_R_LAMP := W#16#0;
   HLINE_DW.SPARE_WORD1 := W#16#0;
   HLINE_DW.SPARE_WORD2 := W#16#0;
   HLINE_DW.SPARE_WORD3 := W#16#0;
   HLINE_DW.SPARE_WORD4 := W#16#0;
   HLINE_DW.S02_LCK1_A_LAMP := W#16#0;
   HLINE_DW.S02_LCK1_R_LAMP := W#16#0;
   HLINE_DW.S02_STP1_A_LAMP := W#16#0;
   HLINE_DW.S02_STP1_R_LAMP := W#16#0;
   HLINE_DW.S02_LCK2_A_LAMP := W#16#0;
   HLINE_DW.S02_LCK2_R_LAMP := W#16#0;
   HLINE_DW.S02_STP2_A_LAMP := W#16#0;
   HLINE_DW.S02_STP2_R_LAMP := W#16#0;
   HLINE_DW.S02_LCK3_A_LAMP := W#16#0;
   HLINE_DW.S02_LCK3_R_LAMP := W#16#0;
   HLINE_DW.S02_STP3_A_LAMP := W#16#0;
   HLINE_DW.S02_STP3_R_LAMP := W#16#0;
   HLINE_DW.S02_ELE_A_LAMP := W#16#0;
   HLINE_DW.S02_ELE_R_LAMP := W#16#0;
   HLINE_DW.S02_RC_A_LAMP := W#16#0;
   HLINE_DW.S02_RC_R_LAMP := W#16#0;
   HLINE_DW.SPARE_WORD15 := W#16#0;
   HLINE_DW.SPARE_WORD16 := W#16#0;
   HLINE_DW.SPARE_WORD17 := W#16#0;
   HLINE_DW.SPARE_WORD18 := W#16#0;
   HLINE_DW.S03_LCK1_A_LAMP := W#16#0;
   HLINE_DW.S03_LCK1_R_LAMP := W#16#0;
   HLINE_DW.S03_STP1_A_LAMP := W#16#0;
   HLINE_DW.S03_STP1_R_LAMP := W#16#0;
   HLINE_DW.S03_ELE_A_LAMP := W#16#0;
   HLINE_DW.S03_ELE_R_LAMP := W#16#0;
   HLINE_DW.SPARE_WORD25 := W#16#0;
   HLINE_DW.SPARE_WORD26 := W#16#0;
   HLINE_DW.SPARE_WORD27 := W#16#0;
   HLINE_DW.SPARE_WORD28 := W#16#0;
   HLINE_DW.RC2_LCK1_A_LAMP := W#16#0;
   HLINE_DW.RC2_LCK1_R_LAMP := W#16#0;
   HLINE_DW.RC2_STP1_A_LAMP := W#16#0;
   HLINE_DW.RC2_STP1_R_LAMP := W#16#0;
   HLINE_DW.RC2_LCK2_A_LAMP := W#16#0;
   HLINE_DW.RC2_LCK2_R_LAMP := W#16#0;
   HLINE_DW.RC2_STP2_A_LAMP := W#16#0;
   HLINE_DW.RC2_STP2_R_LAMP := W#16#0;
   HLINE_DW.RC2_LCK3_A_LAMP1 := W#16#0;
   HLINE_DW.RC2_LCK3_R_LAMP1 := W#16#0;
   HLINE_DW.RC2_STP3_A_LAMP1 := W#16#0;
   HLINE_DW.RC2_STP3_R_LAMP1 := W#16#0;
   HLINE_DW.RC2_LCK4_A_LAMP1 := W#16#0;
   HLINE_DW.RC2_LCK4_R_LAMP1 := W#16#0;
   HLINE_DW.RC2_STP4_A_LAMP1 := W#16#0;
   HLINE_DW.RC2_STP4_R_LAMP1 := W#16#0;
   HLINE_DW.RC2_RC_A_LAMP1 := W#16#0;
   HLINE_DW.RC2_RC_R_LAMP1 := W#16#0;
   HLINE_DW.SPARE_WORD34 := W#16#0;
   HLINE_DW.SPARE_WORD35 := W#16#0;
   HLINE_DW.SPARE_WORD36 := W#16#0;
   HLINE_DW.SPARE_WORD37 := W#16#0;
   HLINE_DW.BUF1_LCK1_A_LAMP := W#16#0;
   HLINE_DW.BUF1_LCK1_R_LAMP := W#16#0;
   HLINE_DW.BUF1_STP1_A_LAMP := W#16#0;
   HLINE_DW.BUF1_STP1_R_LAMP := W#16#0;
   HLINE_DW.SPARE_WORD42 := W#16#0;
   HLINE_DW.SPARE_WORD43 := W#16#0;
   HLINE_DW.SPARE_WORD44 := W#16#0;
   HLINE_DW.SPARE_WORD45 := W#16#0;
   HLINE_DW.BUF2_LCK1_A_LAMP := W#16#0;
   HLINE_DW.BUF2_LCK1_R_LAMP := W#16#0;
   HLINE_DW.BUF2_STP1_A_LAMP := W#16#0;
   HLINE_DW.BUF2_STP1_R_LAMP := W#16#0;
   HLINE_DW.SPARE_WORD50 := W#16#0;
   HLINE_DW.SPARE_WORD51 := W#16#0;
   HLINE_DW.SPARE_WORD52 := W#16#0;
   HLINE_DW.SPARE_WORD53 := W#16#0;
   HLINE_DW.S04_LCK1_A_LAMP := W#16#0;
   HLINE_DW.S04_LCK1_R_LAMP := W#16#0;
   HLINE_DW.S04_STP1_A_LAMP := W#16#0;
   HLINE_DW.S04_STP2_R_LAMP := W#16#0;
   HLINE_DW.S04_ELE_A_LAMP := W#16#0;
   HLINE_DW.S04_ELE_R_LAMP := W#16#0;
   HLINE_DW.S04_HK_A_LAMP := W#16#0;
   HLINE_DW.S04_HK_R_LAMP := W#16#0;
   HLINE_DW.SPARE_WORD55 := W#16#0;
   HLINE_DW.SPARE_WORD56 := W#16#0;
   HLINE_DW.SPARE_WORD57 := W#16#0;
   HLINE_DW.SPARE_WORD58 := W#16#0;
   HLINE_DW.S05_LCK1_A_LAMP := W#16#0;
   HLINE_DW.S05_LCK1_R_LAMP := W#16#0;
   HLINE_DW.S05_STP1_A_LAMP := W#16#0;
   HLINE_DW.S05_STP2_R_LAMP := W#16#0;
   HLINE_DW.S05_ELE_A_LAMP := W#16#0;
   HLINE_DW.S05_ELE_R_LAMP := W#16#0;
   HLINE_DW.S05_HK_A_LAMP := W#16#0;
   HLINE_DW.S05_HK_R_LAMP := W#16#0;
   HLINE_DW.SPARE_WORD60 := W#16#0;
   HLINE_DW.SPARE_WORD61 := W#16#0;
   HLINE_DW.SPARE_WORD62 := W#16#0;
   HLINE_DW.SPARE_WORD63 := W#16#0;
   HLINE_DW.TT_PLOCK_A_LAMP := W#16#0;
   HLINE_DW.TT_PLOCK_R_LAMP := W#16#0;
   HLINE_DW.TT_ELE_A_LAMP := W#16#0;
   HLINE_DW.TT_ELE_R_LAMP := W#16#0;
   HLINE_DW.TT_ROLL_A_LAMP := W#16#0;
   HLINE_DW.TT_ROLL_R_LAMP := W#16#0;
   HLINE_DW.SPARE_WORD70 := W#16#0;
   HLINE_DW.SPARE_WORD71 := W#16#0;
   HLINE_DW.SPARE_WORD72 := W#16#0;
   HLINE_DW.SPARE_WORD73 := W#16#0;
   HLINE_DW.SPARE_WORD74 := W#16#0;
   HLINE_DW.SPARE_WORD75 := W#16#0;
   HLINE_DW.SPARE_WORD76 := W#16#0;
   HLINE_DW.SPARE_WORD77 := W#16#0;
   HLINE_DW.SPARE_WORD78 := W#16#0;
   HLINE_DW.SPARE_WORD79 := W#16#0;
   HLINE_DW.SPARE_WORD80 := W#16#0;
   HLINE_DW.SPARE_WORD81 := W#16#0;
   HLINE_DW.SPARE_WORD82 := W#16#0;
   HLINE_DW.SPARE_WORD83 := W#16#0;
   HLINE_DW.SPARE_WORD84 := W#16#0;
   HLINE_DW.SPARE_WORD85 := W#16#0;
   HLINE_DW.SPARE_WORD86 := W#16#0;
   HLINE_DW.SPARE_WORD87 := W#16#0;
   HLINE_DW.SPARE_WORD88 := W#16#0;
   HLINE_DW.SPARE_WORD89 := W#16#0;
   HLINE_DW.SPARE_WORD90 := W#16#0;
   HLINE_DW.SPARE_WORD91 := W#16#0;
   HLINE_DW.SPARE_WORD92 := W#16#0;
   HLINE_DW.SPARE_WORD93 := W#16#0;
   HLINE_DW.SPARE_WORD94 := W#16#0;
   HLINE_DW.SPARE_WORD95 := W#16#0;
   HLINE_DW.SPARE_WORD96 := W#16#0;
   HLINE_DW.SPARE_WORD97 := W#16#0;
   HLINE_DW.SPARE_WORD98 := W#16#0;
   HLINE_DW.SPARE_WORD99 := W#16#0;
   HLINE_DW.SPARE_WORD100 := W#16#0;
   HLINE_DW.SPARE_WORD101 := W#16#0;
   HLINE_DW.SPARE_WORD102 := W#16#0;
   HLINE_DW.SPARE_WORD103 := W#16#0;
   HLINE_DW.SPARE_WORD104 := W#16#0;
   HLINE_DW.SPARE_WORD105 := W#16#0;
   HLINE_DW.SPARE_WORD106 := W#16#0;
   HLINE_DW.SPARE_WORD107 := W#16#0;
   HLINE_DW.SPARE_WORD108 := W#16#0;
   HLINE_DW.SPARE_WORD109 := W#16#0;
   HLINE_DW.SPARE_WORD110 := W#16#0;
   HLINE_DW.SPARE_WORD111 := W#16#0;
   HLINE_DW.SPARE_WORD112 := W#16#0;
   HLINE_DW.SPARE_WORD113 := W#16#0;
   HLINE_DW.SPARE_WORD114 := W#16#0;
   HLINE_DW.SPARE_WORD115 := W#16#0;
   HLINE_DW.SPARE_WORD116 := W#16#0;
   HLINE_DW.SPARE_WORD117 := W#16#0;
   HLINE_DW.SPARE_WORD118 := W#16#0;
   HLINE_DW.SPARE_WORD119 := W#16#0;
   HLINE_DW.SPARE_WORD120 := W#16#0;
   HLINE_DW.SPARE_WORD121 := W#16#0;
   HLINE_DW.SPARE_WORD122 := W#16#0;
   HLINE_DW.SPARE_WORD123 := W#16#0;
   HLINE_DW.SPARE_WORD124 := W#16#0;
   HLINE_DW.SPARE_WORD125 := W#16#0;
   HLINE_DW.SPARE_WORD126 := W#16#0;
   HLINE_DW.SPARE_WORD127 := W#16#0;
   HLINE_DW.SPARE_WORD128 := W#16#0;
   HLINE_DW.SPARE_WORD129 := W#16#0;
   HLINE_DW.SPARE_WORD130 := W#16#0;
   HLINE_DW.SPARE_WORD131 := W#16#0;
   HLINE_DW.SPARE_WORD132 := W#16#0;
   HLINE_DW.SPARE_WORD133 := W#16#0;
   HLINE_DW.SPARE_WORD134 := W#16#0;
   HLINE_DW.SPARE_WORD135 := W#16#0;
   HUPDL_DX._1ST_U_SEL := FALSE;
   HUPDL_DX._2ND_U1_SEL := FALSE;
   HUPDL_DX._2ND_U2_SEL := FALSE;
   HUPDL_DX.SPUSH1_SEL := FALSE;
   HUPDL_DX.LOCKG_SEL := FALSE;
   HUPDL_DX.SPARE1 := FALSE;
   HUPDL_DX.SPARE2 := FALSE;
   HUPDL_DX.SPARE3 := FALSE;
   HUPDL_DX.Q_1ST_PIN_SEL := FALSE;
   HUPDL_DX.Q_2ND_UNIT_SEL := FALSE;
   HUPDL_DX.Q_3RD_UNIT_SEL := FALSE;
   HUPDL_DX.Q_4TH_UNIT_SEL := FALSE;
   HUPDL_DX.SPARE8 := FALSE;
   HUPDL_DX.SPARE9 := FALSE;
   HUPDL_DX.SPARE10 := FALSE;
   HUPDL_DX.SPARE11 := FALSE;
   HUPDL_DX.SPARE12 := FALSE;
   HUPDL_DX.SPARE13 := FALSE;
   HUPDL_DX.SPARE14 := FALSE;
   HUPDL_DX.SPARE15 := FALSE;
   HUPDL_DX.SPARE16 := FALSE;
   HUPDL_DX.SPARE17 := FALSE;
   HUPDL_DX.SPARE18 := FALSE;
   HUPDL_DX.SPARE19 := FALSE;
   HUPDL_DX.SPARE20 := FALSE;
   HUPDL_DX.SPARE21 := FALSE;
   HUPDL_DX.SPARE22 := FALSE;
   HUPDL_DX.SPARE23 := FALSE;
   HUPDL_DX.SPARE24 := FALSE;
   HUPDL_DX.SPARE25 := FALSE;
   HUPDL_DX.PB_ADV := FALSE;
   HUPDL_DX.PB_RET := FALSE;
   HUPDL_DX.BH_1_SEL := FALSE;
   HUPDL_DX.BH_2_SEL := FALSE;
   HUPDL_DX.BH_3_SEL := FALSE;
   HUPDL_DX.BH_4_SEL := FALSE;
   HUPDL_DX.BH_5_SEL := FALSE;
   HUPDL_DX.BH_6_SEL := FALSE;
   HUPDL_DX.BH_7_SEL := FALSE;
   HUPDL_DX.BH_8_SEL := FALSE;
   HUPDL_DX.BH_9_SEL := FALSE;
   HUPDL_DX.BH_10_SEL := FALSE;
   HUPDL_DX.BH_11_SEL := FALSE;
   HUPDL_DX.BH_12_SEL := FALSE;
   HUPDL_DX.BH_13_SEL := FALSE;
   HUPDL_DX.BH_14_SEL := FALSE;
   HUPDL_DX.BH_15_SEL := FALSE;
   HUPDL_DX.BH_16_SEL := FALSE;
   HUPDL_DX.SPARE42 := FALSE;
   HUPDL_DX.SPARE43 := FALSE;
   HUPDL_DX.SPARE44 := FALSE;
   HUPDL_DX.SPARE45 := FALSE;
   HUPDL_DX.SPARE46 := FALSE;
   HUPDL_DX.SPARE47 := FALSE;
   HUPDL_DX.SPARE48 := FALSE;
   HUPDL_DX.SPARE49 := FALSE;
   HUPDL_DX.SPARE50 := FALSE;
   HUPDL_DX.SPARE51 := FALSE;
   HUPDL_DX.SPARE52 := FALSE;
   HUPDL_DX.SPARE53 := FALSE;
   HUPDL_DX.SPARE54 := FALSE;
   HUPDL_DX.SPARE55 := FALSE;
   HUPDL_DX.SPARE56 := FALSE;
   HUPDL_DX.SPARE57 := FALSE;
   HUPDL_DX.VI_1_SEL := FALSE;
   HUPDL_DX.VI_2_SEL := FALSE;
   HUPDL_DX.VI_3_SEL := FALSE;
   HUPDL_DX.VI_4_SEL := FALSE;
   HUPDL_DX.VI_5_SEL := FALSE;
   HUPDL_DX.VI_6_SEL := FALSE;
   HUPDL_DX.VI_7_SEL := FALSE;
   HUPDL_DX.VI_8_SEL := FALSE;
   HUPDL_DX.VI_9_SEL := FALSE;
   HUPDL_DX.VI_10_SEL := FALSE;
   HUPDL_DX.VI_11_SEL := FALSE;
   HUPDL_DX.VI_12_SEL := FALSE;
   HUPDL_DX.VI_13_SEL := FALSE;
   HUPDL_DX.VI_14_SEL := FALSE;
   HUPDL_DX.VI_15_SEL := FALSE;
   HUPDL_DX.VI_16_SEL := FALSE;
   HUPDL_DX.SPARE59 := FALSE;
   HUPDL_DX.SPARE60 := FALSE;
   HUPDL_DX.SPARE61 := FALSE;
   HUPDL_DX.SPARE62 := FALSE;
   HUPDL_DX.SPARE63 := FALSE;
   HUPDL_DX.SPARE64 := FALSE;
   HUPDL_DX.SPARE65 := FALSE;
   HUPDL_DX.SPARE66 := FALSE;
   HUPDL_DX.SPARE67 := FALSE;
   HUPDL_DX.SPARE68 := FALSE;
   HUPDL_DX.SPARE69 := FALSE;
   HUPDL_DX.SPARE70 := FALSE;
   HUPDL_DX.SPARE71 := FALSE;
   HUPDL_DX.SPARE72 := FALSE;
   HUPDL_DX.SPARE73 := FALSE;
   HUPDL_DX.SPARE74 := FALSE;
   HUPDL_DX.SPARE75 := FALSE;
   HUPDL_DX.SPARE76 := FALSE;
   HUPDL_DX.SPARE77 := FALSE;
   HUPDL_DX.SPARE78 := FALSE;
   HUPDL_DX.SPARE79 := FALSE;
   HUPDL_DX.SPARE80 := FALSE;
   HUPDL_DX.SPARE81 := FALSE;
   HUPDL_DX.SPARE82 := FALSE;
   HUPDL_DX.SPARE83 := FALSE;
   HUPDL_DX.SPARE84 := FALSE;
   HUPDL_DX.SPARE85 := FALSE;
   HUPDL_DX.SPARE86 := FALSE;
   HUPDL_DX.SPARE87 := FALSE;
   HUPDL_DX.SPARE88 := FALSE;
   HUPDL_DX.SPARE89 := FALSE;
   HUPDL_DX.SPARE90 := FALSE;
   HUPDL_DX.SPARE91 := FALSE;
   HUPDL_DX.SPARE92 := FALSE;
   HUPDL_DX.SPARE93 := FALSE;
   HUPDL_DX.SPARE94 := FALSE;
   HUPDL_DX.SPARE95 := FALSE;
   HUPDL_DX.SPARE96 := FALSE;
   HUPDL_DX.SPARE97 := FALSE;
   HUPDL_DX.SPARE98 := FALSE;
   HUPDL_DX.SPARE99 := FALSE;
   HUPDL_DX.SPARE100 := FALSE;
   HUPDL_DX.SPARE101 := FALSE;
   HUPDL_DX.SPARE102 := FALSE;
   HUPDL_DX.SPARE103 := FALSE;
   HUPDL_DX.SPARE104 := FALSE;
   HUPDL_DX.SPARE105 := FALSE;
   HUPDL_DX.SPARE106 := FALSE;
   HUPDL_DX.SPARE107 := FALSE;
   HUPDL_DX.SPARE108 := FALSE;
   HUPDL_DX.SPARE109 := FALSE;
   HUPDL_DX.SPARE110 := FALSE;
   HUPDL_DX.SPARE111 := FALSE;
   HUPDL_DX.SPARE112 := FALSE;
   HUPDL_DX.SPARE113 := FALSE;
   HUPDL_DX.SPARE114 := FALSE;
   HUPDL_DX.SPARE115 := FALSE;
   HUPDL_DX.SPARE116 := FALSE;
   HUPDL_DX.SPARE117 := FALSE;
   HUPDL_DX.SPARE118 := FALSE;
   HUPDL_DX.SPARE119 := FALSE;
   HUPDL_DX.SPARE120 := FALSE;
   HUPDL_DX.SPARE121 := FALSE;
   HUPDL_DX.SPARE122 := FALSE;
   HUPDL_DX.SPARE123 := FALSE;
   HUPDL_DX.SPARE124 := FALSE;
   HUPDL_DX.SPARE125 := FALSE;
   HUPDL_DX.SPARE126 := FALSE;
   HUPDL_DX.SPARE127 := FALSE;
   HUPDL_DX.SPARE128 := FALSE;
   HUPDL_DX.SPARE129 := FALSE;
   HUPDL_DX.SPARE130 := FALSE;
   HUPDL_DX.SPARE131 := FALSE;
   HUPDL_DX.SPARE132 := FALSE;
   HUPDL_DX.SPARE133 := FALSE;
   HUPDL_DX.SPARE134 := FALSE;
   HUPDL_DX.SPARE135 := FALSE;
   HUPDL_DX.SPARE136 := FALSE;
   HUPDL_DX.SPARE137 := FALSE;
   HUPDL_DX.SPARE138 := FALSE;
   HUPDL_DW._1ST_U_ADV_LAMP := W#16#0;
   HUPDL_DW._1ST_U_RET_LAMP := W#16#0;
   HUPDL_DW._2ND_U1_ADV_LAMP := W#16#0;
   HUPDL_DW._2ND_U1_RET_LAMP := W#16#0;
   HUPDL_DW._2ND_U2_ADV_LAMP := W#16#0;
   HUPDL_DW._2ND_U2_RET_LAMP := W#16#0;
   HUPDL_DW.SPUSH1_ADV_LAMP := W#16#0;
   HUPDL_DW.SPUSH1_RET_LAMP := W#16#0;
   HUPDL_DW.LOCKG_ADV_LAMP := W#16#0;
   HUPDL_DW.LOCKG_RET_LAMP := W#16#0;
   HUPDL_DW.SPARE_WORD2 := W#16#0;
   HUPDL_DW.SPARE_WORD3 := W#16#0;
   HUPDL_DW.SPARE_WORD4 := W#16#0;
   HUPDL_DW.SPARE_WORD5 := W#16#0;
   HUPDL_DW.SPARE_WORD6 := W#16#0;
   HUPDL_DW.SPARE_WORD7 := W#16#0;
   HUPDL_DW.SPARE_WORD8 := W#16#0;
   HUPDL_DW.SPARE_WORD9 := W#16#0;
   HUPDL_DW.SPARE_WORD10 := W#16#0;
   HUPDL_DW.SPARE_WORD11 := W#16#0;
   HUPDL_DW.Q_1ST_PIN_ADV_LAMP := W#16#0;
   HUPDL_DW.Q_1ST_PIN_RET_LAMP := W#16#0;
   HUPDL_DW.Q_2ND_UNIT_ADV_LAMP := W#16#0;
   HUPDL_DW.Q_2ND_UNIT_RET_LAMP := W#16#0;
   HUPDL_DW.Q_3RD_UNIT_ADV_LAMP := W#16#0;
   HUPDL_DW.Q_3RD_UNIT_RET_LAMP := W#16#0;
   HUPDL_DW.Q_4TH_UNIT_ADV_LAMP := W#16#0;
   HUPDL_DW.Q_4TH_UNIT_RET_LAMP := W#16#0;
   HUPDL_DW.SPARE_WORD20 := W#16#0;
   HUPDL_DW.SPARE_WORD21 := W#16#0;
   HUPDL_DW.SPARE_WORD22 := W#16#0;
   HUPDL_DW.SPARE_WORD23 := W#16#0;
   HUPDL_DW.BH_1_ADV_LAMP := W#16#0;
   HUPDL_DW.BH_1_RET_LAMP := W#16#0;
   HUPDL_DW.BH_2_ADV_LAMP := W#16#0;
   HUPDL_DW.BH_2_RET_LAMP := W#16#0;
   HUPDL_DW.BH_3_ADV_LAMP := W#16#0;
   HUPDL_DW.BH_3_RET_LAMP := W#16#0;
   HUPDL_DW.BH_4_ADV_LAMP := W#16#0;
   HUPDL_DW.BH_4_RET_LAMP := W#16#0;
   HUPDL_DW.BH_5_ADV_LAMP := W#16#0;
   HUPDL_DW.BH_5_RET_LAMP := W#16#0;
   HUPDL_DW.BH_6_ADV_LAMP := W#16#0;
   HUPDL_DW.BH_6_RET_LAMP := W#16#0;
   HUPDL_DW.BH_7_ADV_LAMP := W#16#0;
   HUPDL_DW.BH_7_RET_LAMP := W#16#0;
   HUPDL_DW.BH_8_ADV_LAMP := W#16#0;
   HUPDL_DW.BH_8_RET_LAMP := W#16#0;
   HUPDL_DW.BH_9_ADV_LAMP := W#16#0;
   HUPDL_DW.BH_9_RET_LAMP := W#16#0;
   HUPDL_DW.BH_10_ADV_LAMP := W#16#0;
   HUPDL_DW.BH_10_RET_LAMP := W#16#0;
   HUPDL_DW.SPARE_WORD54 := W#16#0;
   HUPDL_DW.SPARE_WORD55 := W#16#0;
   HUPDL_DW.SPARE_WORD56 := W#16#0;
   HUPDL_DW.SPARE_WORD57 := W#16#0;
   HUPDL_DW.SPARE_WORD58 := W#16#0;
   HUPDL_DW.SPARE_WORD59 := W#16#0;
   HUPDL_DW.SPARE_WORD60 := W#16#0;
   HUPDL_DW.SPARE_WORD61 := W#16#0;
   HUPDL_DW.SPARE_WORD62 := W#16#0;
   HUPDL_DW.SPARE_WORD63 := W#16#0;
   HUPDL_DW.SPARE_WORD64 := W#16#0;
   HUPDL_DW.SPARE_WORD65 := W#16#0;
   HUPDL_DW.SPARE_WORD66 := W#16#0;
   HUPDL_DW.SPARE_WORD67 := W#16#0;
   HUPDL_DW.SPARE_WORD68 := W#16#0;
   HUPDL_DW.SPARE_WORD69 := W#16#0;
   HUPDL_DW.SPARE_WORD70 := W#16#0;
   HUPDL_DW.SPARE_WORD71 := W#16#0;
   HUPDL_DW.SPARE_WORD72 := W#16#0;
   HUPDL_DW.SPARE_WORD73 := W#16#0;
   HUPDL_DW.SPARE_WORD74 := W#16#0;
   HUPDL_DW.SPARE_WORD75 := W#16#0;
   HUPDL_DW.SPARE_WORD76 := W#16#0;
   HUPDL_DW.SPARE_WORD77 := W#16#0;
   HUPDL_DW.SPARE_WORD78 := W#16#0;
   HUPDL_DW.SPARE_WORD79 := W#16#0;
   HUPDL_DW.SPARE_WORD80 := W#16#0;
   HUPDL_DW.SPARE_WORD81 := W#16#0;
   HUPDL_DW.SPARE_WORD82 := W#16#0;
   HUPDL_DW.SPARE_WORD83 := W#16#0;
   HUPDL_DW.SPARE_WORD84 := W#16#0;
   HUPDL_DW.SPARE_WORD85 := W#16#0;
   HUPDL_DW.SPARE_WORD86 := W#16#0;
   HUPDL_DW.SPARE_WORD87 := W#16#0;
   HUPDL_DW.SPARE_WORD88 := W#16#0;
   HUPDL_DW.SPARE_WORD89 := W#16#0;
   HUPDL_DW.SPARE_WORD90 := W#16#0;
   HUPDL_DW.SPARE_WORD91 := W#16#0;
   HUPDL_DW.SPARE_WORD92 := W#16#0;
   HUPDL_DW.SPARE_WORD93 := W#16#0;
   HUPDL_DW.SPARE_WORD94 := W#16#0;
   HUPDL_DW.SPARE_WORD95 := W#16#0;
   HUPDL_DW.SPARE_WORD96 := W#16#0;
   HUPDL_DW.SPARE_WORD97 := W#16#0;
   HUPDL_DW.SPARE_WORD98 := W#16#0;
   HUPDL_DW.SPARE_WORD99 := W#16#0;
   HUPDL_DW.SPARE_WORD100 := W#16#0;
   HUPDL_DW.SPARE_WORD101 := W#16#0;
   HUPDL_DW.SPARE_WORD102 := W#16#0;
   HUPDL_DW.SPARE_WORD103 := W#16#0;
   HUPDL_DW.SPARE_WORD104 := W#16#0;
   HUPDL_DW.SPARE_WORD105 := W#16#0;
   HUPDL_DW.SPARE_WORD106 := W#16#0;
   HUPDL_DW.SPARE_WORD107 := W#16#0;
   HUPDL_DW.SPARE_WORD108 := W#16#0;
   HUPDL_DW.SPARE_WORD109 := W#16#0;
   HUPDL_DW.SPARE_WORD110 := W#16#0;
   HUPDL_DW.SPARE_WORD111 := W#16#0;
   HUPDL_DW.SPARE_WORD112 := W#16#0;
   HUPDL_DW.SPARE_WORD113 := W#16#0;
   HUPDL_DW.SPARE_WORD114 := W#16#0;
   HUPDL_DW.SPARE_WORD115 := W#16#0;
   HUPDL_DW.SPARE_WORD116 := W#16#0;
   HUPDL_DW.SPARE_WORD117 := W#16#0;
   HUPDL_DW.SPARE_WORD118 := W#16#0;
   HUPDL_DW.SPARE_WORD119 := W#16#0;
   HUPDL_DW.SPARE_WORD120 := W#16#0;
   HUPDL_DW.SPARE_WORD121 := W#16#0;
   HUPDL_DW.SPARE_WORD122 := W#16#0;
   HUPDL_DW.SPARE_WORD123 := W#16#0;
   HUPDL_DW.SPARE_WORD124 := W#16#0;
   HUPDL_DW.SPARE_WORD125 := W#16#0;
   HUPDL_DW.SPARE_WORD126 := W#16#0;
   HUPDL_DW.SPARE_WORD127 := W#16#0;
   HUPDL_DW.SPARE_WORD128 := W#16#0;
   HUPDL_DW.SPARE_WORD129 := W#16#0;
   HUPDL_DW.SPARE_WORD130 := W#16#0;
   HUPDL_DW.SPARE_WORD131 := W#16#0;
   HUPDL_DW.SPARE_WORD132 := W#16#0;
   HUPDL_DW.SPARE_WORD133 := W#16#0;
   HUPDL_DW.SPARE_WORD134 := W#16#0;
   HUPDL_DW.SPARE_WORD135 := W#16#0;
   HUPDL_DW.SPARE_WORD136 := W#16#0;
   HUPDL_DW.SPARE_WORD137 := W#16#0;
   HUPDL_DW.SPARE_WORD138 := W#16#0;
   HUPDL_DW.SPARE_WORD139 := W#16#0;
   HUPDL_DW.SPARE_WORD140 := W#16#0;
   HUPDL_DW.SPARE_WORD141 := W#16#0;
   HUPDL_DW.SPARE_WORD142 := W#16#0;
   HUPDL_DW.SPARE_WORD143 := W#16#0;
   HUPDL_DW.SPARE_WORD144 := W#16#0;
   HUPDL_DW.SPARE_WORD145 := W#16#0;
   HUPDL_DW.SPARE_WORD146 := W#16#0;
   HUPDL_DW.SPARE_WORD147 := W#16#0;
   HUPDL_DW.SPARE_WORD148 := W#16#0;
   HUPDL_DW.SPARE_WORD149 := W#16#0;
   HUPDL_DW.SPARE_WORD150 := W#16#0;
   HUPDL_DW.SPARE_WORD151 := W#16#0;
   HUPDL_DW.SPARE_WORD152 := W#16#0;
   HUPDL_DW.SPARE_WORD153 := W#16#0;
   HUPDL_DW.SPARE_WORD154 := W#16#0;
   HUPDL_DW.SPARE_WORD155 := W#16#0;
   HUPDL_DW.SPARE_WORD156 := W#16#0;
   HUPDL_DW.SPARE_WORD157 := W#16#0;
   HUPDL_DW.SPARE_WORD158 := W#16#0;
   HUPDL_DW.SPARE_WORD159 := W#16#0;
   HUPDL_DW.SPARE_WORD160 := W#16#0;
   HUPDL_DW.SPARE_WORD161 := W#16#0;
   HUPDL_DW.SPARE_WORD162 := W#16#0;
   HUPDL_DW.SPARE_WORD163 := W#16#0;
   HUPDL_DW.SPARE_WORD164 := W#16#0;
   HUPDL_DW.SPARE_WORD165 := W#16#0;
   HUPDL_DW.SPARE_WORD166 := W#16#0;
   HUPDL_DW.SPARE_WORD167 := W#16#0;
   HUPDL_DW.SPARE_WORD168 := W#16#0;
   HUPDL_DW.SPARE_WORD169 := W#16#0;
   HUPDL_DW.SPARE_WORD170 := W#16#0;
   HUPDL_DW.SPARE_WORD171 := W#16#0;
   HUPDL_DW.SPARE_WORD172 := W#16#0;
   HUPDL_DW.SPARE_WORD173 := W#16#0;
   HUPDL_DW.SPARE_WORD174 := W#16#0;
   HUPDL_DW.SPARE_WORD175 := W#16#0;
   HUPDL_DW.SPARE_WORD176 := W#16#0;
   HUPDL_DW.SPARE_WORD177 := W#16#0;
   HUPDL_DW.SPARE_WORD178 := W#16#0;
   HUPDL_DW.SPARE_WORD179 := W#16#0;
   HUPDL_DW.SPARE_WORD180 := W#16#0;
   HUPDL_DW.SPARE_WORD181 := W#16#0;
END_DATA_BLOCK

DATA_BLOCK DB 98
VERSION : 0.1


  STRUCT
   STAT0 : ARRAY  [0 .. 25 ] OF DWORD ;
  END_STRUCT ;
BEGIN
   STAT0[0] := DW#16#0;
   STAT0[1] := DW#16#0;
   STAT0[2] := DW#16#0;
   STAT0[3] := DW#16#0;
   STAT0[4] := DW#16#0;
   STAT0[5] := DW#16#0;
   STAT0[6] := DW#16#0;
   STAT0[7] := DW#16#0;
   STAT0[8] := DW#16#0;
   STAT0[9] := DW#16#0;
   STAT0[10] := DW#16#0;
   STAT0[11] := DW#16#0;
   STAT0[12] := DW#16#0;
   STAT0[13] := DW#16#0;
   STAT0[14] := DW#16#0;
   STAT0[15] := DW#16#0;
   STAT0[16] := DW#16#0;
   STAT0[17] := DW#16#0;
   STAT0[18] := DW#16#0;
   STAT0[19] := DW#16#0;
   STAT0[20] := DW#16#0;
   STAT0[21] := DW#16#0;
   STAT0[22] := DW#16#0;
   STAT0[23] := DW#16#0;
   STAT0[24] := DW#16#0;
   STAT0[25] := DW#16#0;
END_DATA_BLOCK

DATA_BLOCK DB 99
VERSION : 0.1


  STRUCT
   STAT0 : WORD ;
   STAT1 : WORD ;
   STAT2 : WORD ;
   STAT3 : WORD ;
   STAT4 : WORD ;
   STAT5 : WORD ;
   STAT6 : WORD ;
   STAT7 : WORD ;
   STAT8 : WORD ;
   STAT9 : WORD ;
   STAT10 : WORD ;
   STAT11 : WORD ;
   STAT12 : WORD ;
   STAT13 : WORD ;
   STAT14 : WORD ;
   STAT15 : WORD ;
   STAT16 : WORD ;
   STAT17 : WORD ;
   STAT18 : WORD ;
   STAT19 : WORD ;
   STAT20 : WORD ;
   STAT21 : WORD ;
   STAT22 : WORD ;
   STAT23 : WORD ;
   STAT24 : WORD ;
   STAT25 : WORD ;
   STAT26 : WORD ;
   STAT27 : WORD ;
   STAT28 : WORD ;
   STAT29 : WORD ;
   STAT30 : WORD ;
   STAT31 : WORD ;
   STAT32 : WORD ;
   STAT33 : WORD ;
   STAT34 : WORD ;
   STAT35 : WORD ;
   STAT36 : WORD ;
   STAT37 : WORD ;
   STAT38 : WORD ;
   STAT39 : WORD ;
   STAT40 : WORD ;
   STAT41 : WORD ;
   STAT42 : WORD ;
   STAT43 : WORD ;
   STAT44 : WORD ;
   STAT45 : WORD ;
   STAT46 : WORD ;
   STAT47 : WORD ;
   STAT48 : WORD ;
   STAT49 : WORD ;
   STAT50 : WORD ;
   STAT51 : WORD ;
   STAT52 : WORD ;
   STAT53 : WORD ;
   STAT54 : WORD ;
   STAT55 : WORD ;
   STAT56 : WORD ;
   STAT57 : WORD ;
   STAT58 : WORD ;
   STAT59 : WORD ;
   STAT60 : WORD ;
   STAT61 : WORD ;
   STAT62 : WORD ;
   STAT63 : WORD ;
  END_STRUCT ;
BEGIN
   STAT0 := W#16#4101;
   STAT1 := W#16#9000;
   STAT2 := W#16#800;
   STAT3 := W#16#0;
   STAT4 := W#16#4102;
   STAT5 := W#16#9000;
   STAT6 := W#16#800;
   STAT7 := W#16#0;
   STAT8 := W#16#4201;
   STAT9 := W#16#5000;
   STAT10 := W#16#800;
   STAT11 := W#16#0;
   STAT12 := W#16#4102;
   STAT13 := W#16#9000;
   STAT14 := W#16#800;
   STAT15 := W#16#0;
   STAT16 := W#16#4101;
   STAT17 := W#16#9000;
   STAT18 := W#16#800;
   STAT19 := W#16#0;
   STAT20 := W#16#4101;
   STAT21 := W#16#9000;
   STAT22 := W#16#800;
   STAT23 := W#16#0;
   STAT24 := W#16#0;
   STAT25 := W#16#0;
   STAT26 := W#16#0;
   STAT27 := W#16#0;
   STAT28 := W#16#0;
   STAT29 := W#16#0;
   STAT30 := W#16#0;
   STAT31 := W#16#0;
   STAT32 := W#16#0;
   STAT33 := W#16#0;
   STAT34 := W#16#0;
   STAT35 := W#16#0;
   STAT36 := W#16#0;
   STAT37 := W#16#0;
   STAT38 := W#16#0;
   STAT39 := W#16#0;
   STAT40 := W#16#0;
   STAT41 := W#16#0;
   STAT42 := W#16#0;
   STAT43 := W#16#0;
   STAT44 := W#16#0;
   STAT45 := W#16#4102;
   STAT46 := W#16#9000;
   STAT47 := W#16#4201;
   STAT48 := W#16#5000;
   STAT49 := W#16#4102;
   STAT50 := W#16#9000;
   STAT51 := W#16#4201;
   STAT52 := W#16#5000;
   STAT53 := W#16#4101;
   STAT54 := W#16#9000;
   STAT55 := W#16#800;
   STAT56 := W#16#0;
   STAT57 := W#16#0;
   STAT58 := W#16#0;
   STAT59 := W#16#0;
   STAT60 := W#16#0;
   STAT61 := W#16#0;
   STAT62 := W#16#0;
   STAT63 := W#16#0;
END_DATA_BLOCK

DATA_BLOCK DB 325
TITLE =
VERSION : 0.1


  STRUCT
   DP_DIAG1 : ARRAY  [1 .. 100 ] OF BYTE ;
   DP_DIAG2 : ARRAY  [1 .. 100 ] OF BYTE ;
   DP_DIAG3 : ARRAY  [1 .. 100 ] OF BYTE ;
   DP_DIAG4 : ARRAY  [1 .. 100 ] OF BYTE ;
   DP_DIAG5 : ARRAY  [1 .. 100 ] OF BYTE ;
   DP_DIAG6 : ARRAY  [1 .. 100 ] OF BYTE ;
   DP_DIAG7 : ARRAY  [1 .. 100 ] OF BYTE ;
   DP_DIAG8 : ARRAY  [1 .. 100 ] OF BYTE ;
   DP_DIAG9 : ARRAY  [1 .. 100 ] OF BYTE ;
   DP_DIAG10 : ARRAY  [1 .. 100 ] OF BYTE ;
  END_STRUCT ;
BEGIN
   DP_DIAG1[1] := B#16#0;
   DP_DIAG1[2] := B#16#0;
   DP_DIAG1[3] := B#16#0;
   DP_DIAG1[4] := B#16#0;
   DP_DIAG1[5] := B#16#0;
   DP_DIAG1[6] := B#16#0;
   DP_DIAG1[7] := B#16#0;
   DP_DIAG1[8] := B#16#0;
   DP_DIAG1[9] := B#16#0;
   DP_DIAG1[10] := B#16#0;
   DP_DIAG1[11] := B#16#0;
   DP_DIAG1[12] := B#16#0;
   DP_DIAG1[13] := B#16#0;
   DP_DIAG1[14] := B#16#0;
   DP_DIAG1[15] := B#16#0;
   DP_DIAG1[16] := B#16#0;
   DP_DIAG1[17] := B#16#0;
   DP_DIAG1[18] := B#16#0;
   DP_DIAG1[19] := B#16#0;
   DP_DIAG1[20] := B#16#0;
   DP_DIAG1[21] := B#16#0;
   DP_DIAG1[22] := B#16#0;
   DP_DIAG1[23] := B#16#0;
   DP_DIAG1[24] := B#16#0;
   DP_DIAG1[25] := B#16#0;
   DP_DIAG1[26] := B#16#0;
   DP_DIAG1[27] := B#16#0;
   DP_DIAG1[28] := B#16#0;
   DP_DIAG1[29] := B#16#0;
   DP_DIAG1[30] := B#16#0;
   DP_DIAG1[31] := B#16#0;
   DP_DIAG1[32] := B#16#0;
   DP_DIAG1[33] := B#16#0;
   DP_DIAG1[34] := B#16#0;
   DP_DIAG1[35] := B#16#0;
   DP_DIAG1[36] := B#16#0;
   DP_DIAG1[37] := B#16#0;
   DP_DIAG1[38] := B#16#0;
   DP_DIAG1[39] := B#16#0;
   DP_DIAG1[40] := B#16#0;
   DP_DIAG1[41] := B#16#0;
   DP_DIAG1[42] := B#16#0;
   DP_DIAG1[43] := B#16#0;
   DP_DIAG1[44] := B#16#0;
   DP_DIAG1[45] := B#16#0;
   DP_DIAG1[46] := B#16#0;
   DP_DIAG1[47] := B#16#0;
   DP_DIAG1[48] := B#16#0;
   DP_DIAG1[49] := B#16#0;
   DP_DIAG1[50] := B#16#0;
   DP_DIAG1[51] := B#16#0;
   DP_DIAG1[52] := B#16#0;
   DP_DIAG1[53] := B#16#0;
   DP_DIAG1[54] := B#16#0;
   DP_DIAG1[55] := B#16#0;
   DP_DIAG1[56] := B#16#0;
   DP_DIAG1[57] := B#16#0;
   DP_DIAG1[58] := B#16#0;
   DP_DIAG1[59] := B#16#0;
   DP_DIAG1[60] := B#16#0;
   DP_DIAG1[61] := B#16#0;
   DP_DIAG1[62] := B#16#0;
   DP_DIAG1[63] := B#16#0;
   DP_DIAG1[64] := B#16#0;
   DP_DIAG1[65] := B#16#0;
   DP_DIAG1[66] := B#16#0;
   DP_DIAG1[67] := B#16#0;
   DP_DIAG1[68] := B#16#0;
   DP_DIAG1[69] := B#16#0;
   DP_DIAG1[70] := B#16#0;
   DP_DIAG1[71] := B#16#0;
   DP_DIAG1[72] := B#16#0;
   DP_DIAG1[73] := B#16#0;
   DP_DIAG1[74] := B#16#0;
   DP_DIAG1[75] := B#16#0;
   DP_DIAG1[76] := B#16#0;
   DP_DIAG1[77] := B#16#0;
   DP_DIAG1[78] := B#16#0;
   DP_DIAG1[79] := B#16#0;
   DP_DIAG1[80] := B#16#0;
   DP_DIAG1[81] := B#16#0;
   DP_DIAG1[82] := B#16#0;
   DP_DIAG1[83] := B#16#0;
   DP_DIAG1[84] := B#16#0;
   DP_DIAG1[85] := B#16#0;
   DP_DIAG1[86] := B#16#0;
   DP_DIAG1[87] := B#16#0;
   DP_DIAG1[88] := B#16#0;
   DP_DIAG1[89] := B#16#0;
   DP_DIAG1[90] := B#16#0;
   DP_DIAG1[91] := B#16#0;
   DP_DIAG1[92] := B#16#0;
   DP_DIAG1[93] := B#16#0;
   DP_DIAG1[94] := B#16#0;
   DP_DIAG1[95] := B#16#0;
   DP_DIAG1[96] := B#16#0;
   DP_DIAG1[97] := B#16#0;
   DP_DIAG1[98] := B#16#0;
   DP_DIAG1[99] := B#16#0;
   DP_DIAG1[100] := B#16#0;
   DP_DIAG2[1] := B#16#0;
   DP_DIAG2[2] := B#16#0;
   DP_DIAG2[3] := B#16#0;
   DP_DIAG2[4] := B#16#0;
   DP_DIAG2[5] := B#16#0;
   DP_DIAG2[6] := B#16#0;
   DP_DIAG2[7] := B#16#0;
   DP_DIAG2[8] := B#16#0;
   DP_DIAG2[9] := B#16#0;
   DP_DIAG2[10] := B#16#0;
   DP_DIAG2[11] := B#16#0;
   DP_DIAG2[12] := B#16#0;
   DP_DIAG2[13] := B#16#0;
   DP_DIAG2[14] := B#16#0;
   DP_DIAG2[15] := B#16#0;
   DP_DIAG2[16] := B#16#0;
   DP_DIAG2[17] := B#16#0;
   DP_DIAG2[18] := B#16#0;
   DP_DIAG2[19] := B#16#0;
   DP_DIAG2[20] := B#16#0;
   DP_DIAG2[21] := B#16#0;
   DP_DIAG2[22] := B#16#0;
   DP_DIAG2[23] := B#16#0;
   DP_DIAG2[24] := B#16#0;
   DP_DIAG2[25] := B#16#0;
   DP_DIAG2[26] := B#16#0;
   DP_DIAG2[27] := B#16#0;
   DP_DIAG2[28] := B#16#0;
   DP_DIAG2[29] := B#16#0;
   DP_DIAG2[30] := B#16#0;
   DP_DIAG2[31] := B#16#0;
   DP_DIAG2[32] := B#16#0;
   DP_DIAG2[33] := B#16#0;
   DP_DIAG2[34] := B#16#0;
   DP_DIAG2[35] := B#16#0;
   DP_DIAG2[36] := B#16#0;
   DP_DIAG2[37] := B#16#0;
   DP_DIAG2[38] := B#16#0;
   DP_DIAG2[39] := B#16#0;
   DP_DIAG2[40] := B#16#0;
   DP_DIAG2[41] := B#16#0;
   DP_DIAG2[42] := B#16#0;
   DP_DIAG2[43] := B#16#0;
   DP_DIAG2[44] := B#16#0;
   DP_DIAG2[45] := B#16#0;
   DP_DIAG2[46] := B#16#0;
   DP_DIAG2[47] := B#16#0;
   DP_DIAG2[48] := B#16#0;
   DP_DIAG2[49] := B#16#0;
   DP_DIAG2[50] := B#16#0;
   DP_DIAG2[51] := B#16#0;
   DP_DIAG2[52] := B#16#0;
   DP_DIAG2[53] := B#16#0;
   DP_DIAG2[54] := B#16#0;
   DP_DIAG2[55] := B#16#0;
   DP_DIAG2[56] := B#16#0;
   DP_DIAG2[57] := B#16#0;
   DP_DIAG2[58] := B#16#0;
   DP_DIAG2[59] := B#16#0;
   DP_DIAG2[60] := B#16#0;
   DP_DIAG2[61] := B#16#0;
   DP_DIAG2[62] := B#16#0;
   DP_DIAG2[63] := B#16#0;
   DP_DIAG2[64] := B#16#0;
   DP_DIAG2[65] := B#16#0;
   DP_DIAG2[66] := B#16#0;
   DP_DIAG2[67] := B#16#0;
   DP_DIAG2[68] := B#16#0;
   DP_DIAG2[69] := B#16#0;
   DP_DIAG2[70] := B#16#0;
   DP_DIAG2[71] := B#16#0;
   DP_DIAG2[72] := B#16#0;
   DP_DIAG2[73] := B#16#0;
   DP_DIAG2[74] := B#16#0;
   DP_DIAG2[75] := B#16#0;
   DP_DIAG2[76] := B#16#0;
   DP_DIAG2[77] := B#16#0;
   DP_DIAG2[78] := B#16#0;
   DP_DIAG2[79] := B#16#0;
   DP_DIAG2[80] := B#16#0;
   DP_DIAG2[81] := B#16#0;
   DP_DIAG2[82] := B#16#0;
   DP_DIAG2[83] := B#16#0;
   DP_DIAG2[84] := B#16#0;
   DP_DIAG2[85] := B#16#0;
   DP_DIAG2[86] := B#16#0;
   DP_DIAG2[87] := B#16#0;
   DP_DIAG2[88] := B#16#0;
   DP_DIAG2[89] := B#16#0;
   DP_DIAG2[90] := B#16#0;
   DP_DIAG2[91] := B#16#0;
   DP_DIAG2[92] := B#16#0;
   DP_DIAG2[93] := B#16#0;
   DP_DIAG2[94] := B#16#0;
   DP_DIAG2[95] := B#16#0;
   DP_DIAG2[96] := B#16#0;
   DP_DIAG2[97] := B#16#0;
   DP_DIAG2[98] := B#16#0;
   DP_DIAG2[99] := B#16#0;
   DP_DIAG2[100] := B#16#0;
   DP_DIAG3[1] := B#16#0;
   DP_DIAG3[2] := B#16#0;
   DP_DIAG3[3] := B#16#0;
   DP_DIAG3[4] := B#16#0;
   DP_DIAG3[5] := B#16#0;
   DP_DIAG3[6] := B#16#0;
   DP_DIAG3[7] := B#16#0;
   DP_DIAG3[8] := B#16#0;
   DP_DIAG3[9] := B#16#0;
   DP_DIAG3[10] := B#16#0;
   DP_DIAG3[11] := B#16#0;
   DP_DIAG3[12] := B#16#0;
   DP_DIAG3[13] := B#16#0;
   DP_DIAG3[14] := B#16#0;
   DP_DIAG3[15] := B#16#0;
   DP_DIAG3[16] := B#16#0;
   DP_DIAG3[17] := B#16#0;
   DP_DIAG3[18] := B#16#0;
   DP_DIAG3[19] := B#16#0;
   DP_DIAG3[20] := B#16#0;
   DP_DIAG3[21] := B#16#0;
   DP_DIAG3[22] := B#16#0;
   DP_DIAG3[23] := B#16#0;
   DP_DIAG3[24] := B#16#0;
   DP_DIAG3[25] := B#16#0;
   DP_DIAG3[26] := B#16#0;
   DP_DIAG3[27] := B#16#0;
   DP_DIAG3[28] := B#16#0;
   DP_DIAG3[29] := B#16#0;
   DP_DIAG3[30] := B#16#0;
   DP_DIAG3[31] := B#16#0;
   DP_DIAG3[32] := B#16#0;
   DP_DIAG3[33] := B#16#0;
   DP_DIAG3[34] := B#16#0;
   DP_DIAG3[35] := B#16#0;
   DP_DIAG3[36] := B#16#0;
   DP_DIAG3[37] := B#16#0;
   DP_DIAG3[38] := B#16#0;
   DP_DIAG3[39] := B#16#0;
   DP_DIAG3[40] := B#16#0;
   DP_DIAG3[41] := B#16#0;
   DP_DIAG3[42] := B#16#0;
   DP_DIAG3[43] := B#16#0;
   DP_DIAG3[44] := B#16#0;
   DP_DIAG3[45] := B#16#0;
   DP_DIAG3[46] := B#16#0;
   DP_DIAG3[47] := B#16#0;
   DP_DIAG3[48] := B#16#0;
   DP_DIAG3[49] := B#16#0;
   DP_DIAG3[50] := B#16#0;
   DP_DIAG3[51] := B#16#0;
   DP_DIAG3[52] := B#16#0;
   DP_DIAG3[53] := B#16#0;
   DP_DIAG3[54] := B#16#0;
   DP_DIAG3[55] := B#16#0;
   DP_DIAG3[56] := B#16#0;
   DP_DIAG3[57] := B#16#0;
   DP_DIAG3[58] := B#16#0;
   DP_DIAG3[59] := B#16#0;
   DP_DIAG3[60] := B#16#0;
   DP_DIAG3[61] := B#16#0;
   DP_DIAG3[62] := B#16#0;
   DP_DIAG3[63] := B#16#0;
   DP_DIAG3[64] := B#16#0;
   DP_DIAG3[65] := B#16#0;
   DP_DIAG3[66] := B#16#0;
   DP_DIAG3[67] := B#16#0;
   DP_DIAG3[68] := B#16#0;
   DP_DIAG3[69] := B#16#0;
   DP_DIAG3[70] := B#16#0;
   DP_DIAG3[71] := B#16#0;
   DP_DIAG3[72] := B#16#0;
   DP_DIAG3[73] := B#16#0;
   DP_DIAG3[74] := B#16#0;
   DP_DIAG3[75] := B#16#0;
   DP_DIAG3[76] := B#16#0;
   DP_DIAG3[77] := B#16#0;
   DP_DIAG3[78] := B#16#0;
   DP_DIAG3[79] := B#16#0;
   DP_DIAG3[80] := B#16#0;
   DP_DIAG3[81] := B#16#0;
   DP_DIAG3[82] := B#16#0;
   DP_DIAG3[83] := B#16#0;
   DP_DIAG3[84] := B#16#0;
   DP_DIAG3[85] := B#16#0;
   DP_DIAG3[86] := B#16#0;
   DP_DIAG3[87] := B#16#0;
   DP_DIAG3[88] := B#16#0;
   DP_DIAG3[89] := B#16#0;
   DP_DIAG3[90] := B#16#0;
   DP_DIAG3[91] := B#16#0;
   DP_DIAG3[92] := B#16#0;
   DP_DIAG3[93] := B#16#0;
   DP_DIAG3[94] := B#16#0;
   DP_DIAG3[95] := B#16#0;
   DP_DIAG3[96] := B#16#0;
   DP_DIAG3[97] := B#16#0;
   DP_DIAG3[98] := B#16#0;
   DP_DIAG3[99] := B#16#0;
   DP_DIAG3[100] := B#16#0;
   DP_DIAG4[1] := B#16#0;
   DP_DIAG4[2] := B#16#0;
   DP_DIAG4[3] := B#16#0;
   DP_DIAG4[4] := B#16#0;
   DP_DIAG4[5] := B#16#0;
   DP_DIAG4[6] := B#16#0;
   DP_DIAG4[7] := B#16#0;
   DP_DIAG4[8] := B#16#0;
   DP_DIAG4[9] := B#16#0;
   DP_DIAG4[10] := B#16#0;
   DP_DIAG4[11] := B#16#0;
   DP_DIAG4[12] := B#16#0;
   DP_DIAG4[13] := B#16#0;
   DP_DIAG4[14] := B#16#0;
   DP_DIAG4[15] := B#16#0;
   DP_DIAG4[16] := B#16#0;
   DP_DIAG4[17] := B#16#0;
   DP_DIAG4[18] := B#16#0;
   DP_DIAG4[19] := B#16#0;
   DP_DIAG4[20] := B#16#0;
   DP_DIAG4[21] := B#16#0;
   DP_DIAG4[22] := B#16#0;
   DP_DIAG4[23] := B#16#0;
   DP_DIAG4[24] := B#16#0;
   DP_DIAG4[25] := B#16#0;
   DP_DIAG4[26] := B#16#0;
   DP_DIAG4[27] := B#16#0;
   DP_DIAG4[28] := B#16#0;
   DP_DIAG4[29] := B#16#0;
   DP_DIAG4[30] := B#16#0;
   DP_DIAG4[31] := B#16#0;
   DP_DIAG4[32] := B#16#0;
   DP_DIAG4[33] := B#16#0;
   DP_DIAG4[34] := B#16#0;
   DP_DIAG4[35] := B#16#0;
   DP_DIAG4[36] := B#16#0;
   DP_DIAG4[37] := B#16#0;
   DP_DIAG4[38] := B#16#0;
   DP_DIAG4[39] := B#16#0;
   DP_DIAG4[40] := B#16#0;
   DP_DIAG4[41] := B#16#0;
   DP_DIAG4[42] := B#16#0;
   DP_DIAG4[43] := B#16#0;
   DP_DIAG4[44] := B#16#0;
   DP_DIAG4[45] := B#16#0;
   DP_DIAG4[46] := B#16#0;
   DP_DIAG4[47] := B#16#0;
   DP_DIAG4[48] := B#16#0;
   DP_DIAG4[49] := B#16#0;
   DP_DIAG4[50] := B#16#0;
   DP_DIAG4[51] := B#16#0;
   DP_DIAG4[52] := B#16#0;
   DP_DIAG4[53] := B#16#0;
   DP_DIAG4[54] := B#16#0;
   DP_DIAG4[55] := B#16#0;
   DP_DIAG4[56] := B#16#0;
   DP_DIAG4[57] := B#16#0;
   DP_DIAG4[58] := B#16#0;
   DP_DIAG4[59] := B#16#0;
   DP_DIAG4[60] := B#16#0;
   DP_DIAG4[61] := B#16#0;
   DP_DIAG4[62] := B#16#0;
   DP_DIAG4[63] := B#16#0;
   DP_DIAG4[64] := B#16#0;
   DP_DIAG4[65] := B#16#0;
   DP_DIAG4[66] := B#16#0;
   DP_DIAG4[67] := B#16#0;
   DP_DIAG4[68] := B#16#0;
   DP_DIAG4[69] := B#16#0;
   DP_DIAG4[70] := B#16#0;
   DP_DIAG4[71] := B#16#0;
   DP_DIAG4[72] := B#16#0;
   DP_DIAG4[73] := B#16#0;
   DP_DIAG4[74] := B#16#0;
   DP_DIAG4[75] := B#16#0;
   DP_DIAG4[76] := B#16#0;
   DP_DIAG4[77] := B#16#0;
   DP_DIAG4[78] := B#16#0;
   DP_DIAG4[79] := B#16#0;
   DP_DIAG4[80] := B#16#0;
   DP_DIAG4[81] := B#16#0;
   DP_DIAG4[82] := B#16#0;
   DP_DIAG4[83] := B#16#0;
   DP_DIAG4[84] := B#16#0;
   DP_DIAG4[85] := B#16#0;
   DP_DIAG4[86] := B#16#0;
   DP_DIAG4[87] := B#16#0;
   DP_DIAG4[88] := B#16#0;
   DP_DIAG4[89] := B#16#0;
   DP_DIAG4[90] := B#16#0;
   DP_DIAG4[91] := B#16#0;
   DP_DIAG4[92] := B#16#0;
   DP_DIAG4[93] := B#16#0;
   DP_DIAG4[94] := B#16#0;
   DP_DIAG4[95] := B#16#0;
   DP_DIAG4[96] := B#16#0;
   DP_DIAG4[97] := B#16#0;
   DP_DIAG4[98] := B#16#0;
   DP_DIAG4[99] := B#16#0;
   DP_DIAG4[100] := B#16#0;
   DP_DIAG5[1] := B#16#0;
   DP_DIAG5[2] := B#16#0;
   DP_DIAG5[3] := B#16#0;
   DP_DIAG5[4] := B#16#0;
   DP_DIAG5[5] := B#16#0;
   DP_DIAG5[6] := B#16#0;
   DP_DIAG5[7] := B#16#0;
   DP_DIAG5[8] := B#16#0;
   DP_DIAG5[9] := B#16#0;
   DP_DIAG5[10] := B#16#0;
   DP_DIAG5[11] := B#16#0;
   DP_DIAG5[12] := B#16#0;
   DP_DIAG5[13] := B#16#0;
   DP_DIAG5[14] := B#16#0;
   DP_DIAG5[15] := B#16#0;
   DP_DIAG5[16] := B#16#0;
   DP_DIAG5[17] := B#16#0;
   DP_DIAG5[18] := B#16#0;
   DP_DIAG5[19] := B#16#0;
   DP_DIAG5[20] := B#16#0;
   DP_DIAG5[21] := B#16#0;
   DP_DIAG5[22] := B#16#0;
   DP_DIAG5[23] := B#16#0;
   DP_DIAG5[24] := B#16#0;
   DP_DIAG5[25] := B#16#0;
   DP_DIAG5[26] := B#16#0;
   DP_DIAG5[27] := B#16#0;
   DP_DIAG5[28] := B#16#0;
   DP_DIAG5[29] := B#16#0;
   DP_DIAG5[30] := B#16#0;
   DP_DIAG5[31] := B#16#0;
   DP_DIAG5[32] := B#16#0;
   DP_DIAG5[33] := B#16#0;
   DP_DIAG5[34] := B#16#0;
   DP_DIAG5[35] := B#16#0;
   DP_DIAG5[36] := B#16#0;
   DP_DIAG5[37] := B#16#0;
   DP_DIAG5[38] := B#16#0;
   DP_DIAG5[39] := B#16#0;
   DP_DIAG5[40] := B#16#0;
   DP_DIAG5[41] := B#16#0;
   DP_DIAG5[42] := B#16#0;
   DP_DIAG5[43] := B#16#0;
   DP_DIAG5[44] := B#16#0;
   DP_DIAG5[45] := B#16#0;
   DP_DIAG5[46] := B#16#0;
   DP_DIAG5[47] := B#16#0;
   DP_DIAG5[48] := B#16#0;
   DP_DIAG5[49] := B#16#0;
   DP_DIAG5[50] := B#16#0;
   DP_DIAG5[51] := B#16#0;
   DP_DIAG5[52] := B#16#0;
   DP_DIAG5[53] := B#16#0;
   DP_DIAG5[54] := B#16#0;
   DP_DIAG5[55] := B#16#0;
   DP_DIAG5[56] := B#16#0;
   DP_DIAG5[57] := B#16#0;
   DP_DIAG5[58] := B#16#0;
   DP_DIAG5[59] := B#16#0;
   DP_DIAG5[60] := B#16#0;
   DP_DIAG5[61] := B#16#0;
   DP_DIAG5[62] := B#16#0;
   DP_DIAG5[63] := B#16#0;
   DP_DIAG5[64] := B#16#0;
   DP_DIAG5[65] := B#16#0;
   DP_DIAG5[66] := B#16#0;
   DP_DIAG5[67] := B#16#0;
   DP_DIAG5[68] := B#16#0;
   DP_DIAG5[69] := B#16#0;
   DP_DIAG5[70] := B#16#0;
   DP_DIAG5[71] := B#16#0;
   DP_DIAG5[72] := B#16#0;
   DP_DIAG5[73] := B#16#0;
   DP_DIAG5[74] := B#16#0;
   DP_DIAG5[75] := B#16#0;
   DP_DIAG5[76] := B#16#0;
   DP_DIAG5[77] := B#16#0;
   DP_DIAG5[78] := B#16#0;
   DP_DIAG5[79] := B#16#0;
   DP_DIAG5[80] := B#16#0;
   DP_DIAG5[81] := B#16#0;
   DP_DIAG5[82] := B#16#0;
   DP_DIAG5[83] := B#16#0;
   DP_DIAG5[84] := B#16#0;
   DP_DIAG5[85] := B#16#0;
   DP_DIAG5[86] := B#16#0;
   DP_DIAG5[87] := B#16#0;
   DP_DIAG5[88] := B#16#0;
   DP_DIAG5[89] := B#16#0;
   DP_DIAG5[90] := B#16#0;
   DP_DIAG5[91] := B#16#0;
   DP_DIAG5[92] := B#16#0;
   DP_DIAG5[93] := B#16#0;
   DP_DIAG5[94] := B#16#0;
   DP_DIAG5[95] := B#16#0;
   DP_DIAG5[96] := B#16#0;
   DP_DIAG5[97] := B#16#0;
   DP_DIAG5[98] := B#16#0;
   DP_DIAG5[99] := B#16#0;
   DP_DIAG5[100] := B#16#0;
   DP_DIAG6[1] := B#16#0;
   DP_DIAG6[2] := B#16#0;
   DP_DIAG6[3] := B#16#0;
   DP_DIAG6[4] := B#16#0;
   DP_DIAG6[5] := B#16#0;
   DP_DIAG6[6] := B#16#0;
   DP_DIAG6[7] := B#16#0;
   DP_DIAG6[8] := B#16#0;
   DP_DIAG6[9] := B#16#0;
   DP_DIAG6[10] := B#16#0;
   DP_DIAG6[11] := B#16#0;
   DP_DIAG6[12] := B#16#0;
   DP_DIAG6[13] := B#16#0;
   DP_DIAG6[14] := B#16#0;
   DP_DIAG6[15] := B#16#0;
   DP_DIAG6[16] := B#16#0;
   DP_DIAG6[17] := B#16#0;
   DP_DIAG6[18] := B#16#0;
   DP_DIAG6[19] := B#16#0;
   DP_DIAG6[20] := B#16#0;
   DP_DIAG6[21] := B#16#0;
   DP_DIAG6[22] := B#16#0;
   DP_DIAG6[23] := B#16#0;
   DP_DIAG6[24] := B#16#0;
   DP_DIAG6[25] := B#16#0;
   DP_DIAG6[26] := B#16#0;
   DP_DIAG6[27] := B#16#0;
   DP_DIAG6[28] := B#16#0;
   DP_DIAG6[29] := B#16#0;
   DP_DIAG6[30] := B#16#0;
   DP_DIAG6[31] := B#16#0;
   DP_DIAG6[32] := B#16#0;
   DP_DIAG6[33] := B#16#0;
   DP_DIAG6[34] := B#16#0;
   DP_DIAG6[35] := B#16#0;
   DP_DIAG6[36] := B#16#0;
   DP_DIAG6[37] := B#16#0;
   DP_DIAG6[38] := B#16#0;
   DP_DIAG6[39] := B#16#0;
   DP_DIAG6[40] := B#16#0;
   DP_DIAG6[41] := B#16#0;
   DP_DIAG6[42] := B#16#0;
   DP_DIAG6[43] := B#16#0;
   DP_DIAG6[44] := B#16#0;
   DP_DIAG6[45] := B#16#0;
   DP_DIAG6[46] := B#16#0;
   DP_DIAG6[47] := B#16#0;
   DP_DIAG6[48] := B#16#0;
   DP_DIAG6[49] := B#16#0;
   DP_DIAG6[50] := B#16#0;
   DP_DIAG6[51] := B#16#0;
   DP_DIAG6[52] := B#16#0;
   DP_DIAG6[53] := B#16#0;
   DP_DIAG6[54] := B#16#0;
   DP_DIAG6[55] := B#16#0;
   DP_DIAG6[56] := B#16#0;
   DP_DIAG6[57] := B#16#0;
   DP_DIAG6[58] := B#16#0;
   DP_DIAG6[59] := B#16#0;
   DP_DIAG6[60] := B#16#0;
   DP_DIAG6[61] := B#16#0;
   DP_DIAG6[62] := B#16#0;
   DP_DIAG6[63] := B#16#0;
   DP_DIAG6[64] := B#16#0;
   DP_DIAG6[65] := B#16#0;
   DP_DIAG6[66] := B#16#0;
   DP_DIAG6[67] := B#16#0;
   DP_DIAG6[68] := B#16#0;
   DP_DIAG6[69] := B#16#0;
   DP_DIAG6[70] := B#16#0;
   DP_DIAG6[71] := B#16#0;
   DP_DIAG6[72] := B#16#0;
   DP_DIAG6[73] := B#16#0;
   DP_DIAG6[74] := B#16#0;
   DP_DIAG6[75] := B#16#0;
   DP_DIAG6[76] := B#16#0;
   DP_DIAG6[77] := B#16#0;
   DP_DIAG6[78] := B#16#0;
   DP_DIAG6[79] := B#16#0;
   DP_DIAG6[80] := B#16#0;
   DP_DIAG6[81] := B#16#0;
   DP_DIAG6[82] := B#16#0;
   DP_DIAG6[83] := B#16#0;
   DP_DIAG6[84] := B#16#0;
   DP_DIAG6[85] := B#16#0;
   DP_DIAG6[86] := B#16#0;
   DP_DIAG6[87] := B#16#0;
   DP_DIAG6[88] := B#16#0;
   DP_DIAG6[89] := B#16#0;
   DP_DIAG6[90] := B#16#0;
   DP_DIAG6[91] := B#16#0;
   DP_DIAG6[92] := B#16#0;
   DP_DIAG6[93] := B#16#0;
   DP_DIAG6[94] := B#16#0;
   DP_DIAG6[95] := B#16#0;
   DP_DIAG6[96] := B#16#0;
   DP_DIAG6[97] := B#16#0;
   DP_DIAG6[98] := B#16#0;
   DP_DIAG6[99] := B#16#0;
   DP_DIAG6[100] := B#16#0;
   DP_DIAG7[1] := B#16#0;
   DP_DIAG7[2] := B#16#0;
   DP_DIAG7[3] := B#16#0;
   DP_DIAG7[4] := B#16#0;
   DP_DIAG7[5] := B#16#0;
   DP_DIAG7[6] := B#16#0;
   DP_DIAG7[7] := B#16#0;
   DP_DIAG7[8] := B#16#0;
   DP_DIAG7[9] := B#16#0;
   DP_DIAG7[10] := B#16#0;
   DP_DIAG7[11] := B#16#0;
   DP_DIAG7[12] := B#16#0;
   DP_DIAG7[13] := B#16#0;
   DP_DIAG7[14] := B#16#0;
   DP_DIAG7[15] := B#16#0;
   DP_DIAG7[16] := B#16#0;
   DP_DIAG7[17] := B#16#0;
   DP_DIAG7[18] := B#16#0;
   DP_DIAG7[19] := B#16#0;
   DP_DIAG7[20] := B#16#0;
   DP_DIAG7[21] := B#16#0;
   DP_DIAG7[22] := B#16#0;
   DP_DIAG7[23] := B#16#0;
   DP_DIAG7[24] := B#16#0;
   DP_DIAG7[25] := B#16#0;
   DP_DIAG7[26] := B#16#0;
   DP_DIAG7[27] := B#16#0;
   DP_DIAG7[28] := B#16#0;
   DP_DIAG7[29] := B#16#0;
   DP_DIAG7[30] := B#16#0;
   DP_DIAG7[31] := B#16#0;
   DP_DIAG7[32] := B#16#0;
   DP_DIAG7[33] := B#16#0;
   DP_DIAG7[34] := B#16#0;
   DP_DIAG7[35] := B#16#0;
   DP_DIAG7[36] := B#16#0;
   DP_DIAG7[37] := B#16#0;
   DP_DIAG7[38] := B#16#0;
   DP_DIAG7[39] := B#16#0;
   DP_DIAG7[40] := B#16#0;
   DP_DIAG7[41] := B#16#0;
   DP_DIAG7[42] := B#16#0;
   DP_DIAG7[43] := B#16#0;
   DP_DIAG7[44] := B#16#0;
   DP_DIAG7[45] := B#16#0;
   DP_DIAG7[46] := B#16#0;
   DP_DIAG7[47] := B#16#0;
   DP_DIAG7[48] := B#16#0;
   DP_DIAG7[49] := B#16#0;
   DP_DIAG7[50] := B#16#0;
   DP_DIAG7[51] := B#16#0;
   DP_DIAG7[52] := B#16#0;
   DP_DIAG7[53] := B#16#0;
   DP_DIAG7[54] := B#16#0;
   DP_DIAG7[55] := B#16#0;
   DP_DIAG7[56] := B#16#0;
   DP_DIAG7[57] := B#16#0;
   DP_DIAG7[58] := B#16#0;
   DP_DIAG7[59] := B#16#0;
   DP_DIAG7[60] := B#16#0;
   DP_DIAG7[61] := B#16#0;
   DP_DIAG7[62] := B#16#0;
   DP_DIAG7[63] := B#16#0;
   DP_DIAG7[64] := B#16#0;
   DP_DIAG7[65] := B#16#0;
   DP_DIAG7[66] := B#16#0;
   DP_DIAG7[67] := B#16#0;
   DP_DIAG7[68] := B#16#0;
   DP_DIAG7[69] := B#16#0;
   DP_DIAG7[70] := B#16#0;
   DP_DIAG7[71] := B#16#0;
   DP_DIAG7[72] := B#16#0;
   DP_DIAG7[73] := B#16#0;
   DP_DIAG7[74] := B#16#0;
   DP_DIAG7[75] := B#16#0;
   DP_DIAG7[76] := B#16#0;
   DP_DIAG7[77] := B#16#0;
   DP_DIAG7[78] := B#16#0;
   DP_DIAG7[79] := B#16#0;
   DP_DIAG7[80] := B#16#0;
   DP_DIAG7[81] := B#16#0;
   DP_DIAG7[82] := B#16#0;
   DP_DIAG7[83] := B#16#0;
   DP_DIAG7[84] := B#16#0;
   DP_DIAG7[85] := B#16#0;
   DP_DIAG7[86] := B#16#0;
   DP_DIAG7[87] := B#16#0;
   DP_DIAG7[88] := B#16#0;
   DP_DIAG7[89] := B#16#0;
   DP_DIAG7[90] := B#16#0;
   DP_DIAG7[91] := B#16#0;
   DP_DIAG7[92] := B#16#0;
   DP_DIAG7[93] := B#16#0;
   DP_DIAG7[94] := B#16#0;
   DP_DIAG7[95] := B#16#0;
   DP_DIAG7[96] := B#16#0;
   DP_DIAG7[97] := B#16#0;
   DP_DIAG7[98] := B#16#0;
   DP_DIAG7[99] := B#16#0;
   DP_DIAG7[100] := B#16#0;
   DP_DIAG8[1] := B#16#0;
   DP_DIAG8[2] := B#16#0;
   DP_DIAG8[3] := B#16#0;
   DP_DIAG8[4] := B#16#0;
   DP_DIAG8[5] := B#16#0;
   DP_DIAG8[6] := B#16#0;
   DP_DIAG8[7] := B#16#0;
   DP_DIAG8[8] := B#16#0;
   DP_DIAG8[9] := B#16#0;
   DP_DIAG8[10] := B#16#0;
   DP_DIAG8[11] := B#16#0;
   DP_DIAG8[12] := B#16#0;
   DP_DIAG8[13] := B#16#0;
   DP_DIAG8[14] := B#16#0;
   DP_DIAG8[15] := B#16#0;
   DP_DIAG8[16] := B#16#0;
   DP_DIAG8[17] := B#16#0;
   DP_DIAG8[18] := B#16#0;
   DP_DIAG8[19] := B#16#0;
   DP_DIAG8[20] := B#16#0;
   DP_DIAG8[21] := B#16#0;
   DP_DIAG8[22] := B#16#0;
   DP_DIAG8[23] := B#16#0;
   DP_DIAG8[24] := B#16#0;
   DP_DIAG8[25] := B#16#0;
   DP_DIAG8[26] := B#16#0;
   DP_DIAG8[27] := B#16#0;
   DP_DIAG8[28] := B#16#0;
   DP_DIAG8[29] := B#16#0;
   DP_DIAG8[30] := B#16#0;
   DP_DIAG8[31] := B#16#0;
   DP_DIAG8[32] := B#16#0;
   DP_DIAG8[33] := B#16#0;
   DP_DIAG8[34] := B#16#0;
   DP_DIAG8[35] := B#16#0;
   DP_DIAG8[36] := B#16#0;
   DP_DIAG8[37] := B#16#0;
   DP_DIAG8[38] := B#16#0;
   DP_DIAG8[39] := B#16#0;
   DP_DIAG8[40] := B#16#0;
   DP_DIAG8[41] := B#16#0;
   DP_DIAG8[42] := B#16#0;
   DP_DIAG8[43] := B#16#0;
   DP_DIAG8[44] := B#16#0;
   DP_DIAG8[45] := B#16#0;
   DP_DIAG8[46] := B#16#0;
   DP_DIAG8[47] := B#16#0;
   DP_DIAG8[48] := B#16#0;
   DP_DIAG8[49] := B#16#0;
   DP_DIAG8[50] := B#16#0;
   DP_DIAG8[51] := B#16#0;
   DP_DIAG8[52] := B#16#0;
   DP_DIAG8[53] := B#16#0;
   DP_DIAG8[54] := B#16#0;
   DP_DIAG8[55] := B#16#0;
   DP_DIAG8[56] := B#16#0;
   DP_DIAG8[57] := B#16#0;
   DP_DIAG8[58] := B#16#0;
   DP_DIAG8[59] := B#16#0;
   DP_DIAG8[60] := B#16#0;
   DP_DIAG8[61] := B#16#0;
   DP_DIAG8[62] := B#16#0;
   DP_DIAG8[63] := B#16#0;
   DP_DIAG8[64] := B#16#0;
   DP_DIAG8[65] := B#16#0;
   DP_DIAG8[66] := B#16#0;
   DP_DIAG8[67] := B#16#0;
   DP_DIAG8[68] := B#16#0;
   DP_DIAG8[69] := B#16#0;
   DP_DIAG8[70] := B#16#0;
   DP_DIAG8[71] := B#16#0;
   DP_DIAG8[72] := B#16#0;
   DP_DIAG8[73] := B#16#0;
   DP_DIAG8[74] := B#16#0;
   DP_DIAG8[75] := B#16#0;
   DP_DIAG8[76] := B#16#0;
   DP_DIAG8[77] := B#16#0;
   DP_DIAG8[78] := B#16#0;
   DP_DIAG8[79] := B#16#0;
   DP_DIAG8[80] := B#16#0;
   DP_DIAG8[81] := B#16#0;
   DP_DIAG8[82] := B#16#0;
   DP_DIAG8[83] := B#16#0;
   DP_DIAG8[84] := B#16#0;
   DP_DIAG8[85] := B#16#0;
   DP_DIAG8[86] := B#16#0;
   DP_DIAG8[87] := B#16#0;
   DP_DIAG8[88] := B#16#0;
   DP_DIAG8[89] := B#16#0;
   DP_DIAG8[90] := B#16#0;
   DP_DIAG8[91] := B#16#0;
   DP_DIAG8[92] := B#16#0;
   DP_DIAG8[93] := B#16#0;
   DP_DIAG8[94] := B#16#0;
   DP_DIAG8[95] := B#16#0;
   DP_DIAG8[96] := B#16#0;
   DP_DIAG8[97] := B#16#0;
   DP_DIAG8[98] := B#16#0;
   DP_DIAG8[99] := B#16#0;
   DP_DIAG8[100] := B#16#0;
   DP_DIAG9[1] := B#16#0;
   DP_DIAG9[2] := B#16#0;
   DP_DIAG9[3] := B#16#0;
   DP_DIAG9[4] := B#16#0;
   DP_DIAG9[5] := B#16#0;
   DP_DIAG9[6] := B#16#0;
   DP_DIAG9[7] := B#16#0;
   DP_DIAG9[8] := B#16#0;
   DP_DIAG9[9] := B#16#0;
   DP_DIAG9[10] := B#16#0;
   DP_DIAG9[11] := B#16#0;
   DP_DIAG9[12] := B#16#0;
   DP_DIAG9[13] := B#16#0;
   DP_DIAG9[14] := B#16#0;
   DP_DIAG9[15] := B#16#0;
   DP_DIAG9[16] := B#16#0;
   DP_DIAG9[17] := B#16#0;
   DP_DIAG9[18] := B#16#0;
   DP_DIAG9[19] := B#16#0;
   DP_DIAG9[20] := B#16#0;
   DP_DIAG9[21] := B#16#0;
   DP_DIAG9[22] := B#16#0;
   DP_DIAG9[23] := B#16#0;
   DP_DIAG9[24] := B#16#0;
   DP_DIAG9[25] := B#16#0;
   DP_DIAG9[26] := B#16#0;
   DP_DIAG9[27] := B#16#0;
   DP_DIAG9[28] := B#16#0;
   DP_DIAG9[29] := B#16#0;
   DP_DIAG9[30] := B#16#0;
   DP_DIAG9[31] := B#16#0;
   DP_DIAG9[32] := B#16#0;
   DP_DIAG9[33] := B#16#0;
   DP_DIAG9[34] := B#16#0;
   DP_DIAG9[35] := B#16#0;
   DP_DIAG9[36] := B#16#0;
   DP_DIAG9[37] := B#16#0;
   DP_DIAG9[38] := B#16#0;
   DP_DIAG9[39] := B#16#0;
   DP_DIAG9[40] := B#16#0;
   DP_DIAG9[41] := B#16#0;
   DP_DIAG9[42] := B#16#0;
   DP_DIAG9[43] := B#16#0;
   DP_DIAG9[44] := B#16#0;
   DP_DIAG9[45] := B#16#0;
   DP_DIAG9[46] := B#16#0;
   DP_DIAG9[47] := B#16#0;
   DP_DIAG9[48] := B#16#0;
   DP_DIAG9[49] := B#16#0;
   DP_DIAG9[50] := B#16#0;
   DP_DIAG9[51] := B#16#0;
   DP_DIAG9[52] := B#16#0;
   DP_DIAG9[53] := B#16#0;
   DP_DIAG9[54] := B#16#0;
   DP_DIAG9[55] := B#16#0;
   DP_DIAG9[56] := B#16#0;
   DP_DIAG9[57] := B#16#0;
   DP_DIAG9[58] := B#16#0;
   DP_DIAG9[59] := B#16#0;
   DP_DIAG9[60] := B#16#0;
   DP_DIAG9[61] := B#16#0;
   DP_DIAG9[62] := B#16#0;
   DP_DIAG9[63] := B#16#0;
   DP_DIAG9[64] := B#16#0;
   DP_DIAG9[65] := B#16#0;
   DP_DIAG9[66] := B#16#0;
   DP_DIAG9[67] := B#16#0;
   DP_DIAG9[68] := B#16#0;
   DP_DIAG9[69] := B#16#0;
   DP_DIAG9[70] := B#16#0;
   DP_DIAG9[71] := B#16#0;
   DP_DIAG9[72] := B#16#0;
   DP_DIAG9[73] := B#16#0;
   DP_DIAG9[74] := B#16#0;
   DP_DIAG9[75] := B#16#0;
   DP_DIAG9[76] := B#16#0;
   DP_DIAG9[77] := B#16#0;
   DP_DIAG9[78] := B#16#0;
   DP_DIAG9[79] := B#16#0;
   DP_DIAG9[80] := B#16#0;
   DP_DIAG9[81] := B#16#0;
   DP_DIAG9[82] := B#16#0;
   DP_DIAG9[83] := B#16#0;
   DP_DIAG9[84] := B#16#0;
   DP_DIAG9[85] := B#16#0;
   DP_DIAG9[86] := B#16#0;
   DP_DIAG9[87] := B#16#0;
   DP_DIAG9[88] := B#16#0;
   DP_DIAG9[89] := B#16#0;
   DP_DIAG9[90] := B#16#0;
   DP_DIAG9[91] := B#16#0;
   DP_DIAG9[92] := B#16#0;
   DP_DIAG9[93] := B#16#0;
   DP_DIAG9[94] := B#16#0;
   DP_DIAG9[95] := B#16#0;
   DP_DIAG9[96] := B#16#0;
   DP_DIAG9[97] := B#16#0;
   DP_DIAG9[98] := B#16#0;
   DP_DIAG9[99] := B#16#0;
   DP_DIAG9[100] := B#16#0;
   DP_DIAG10[1] := B#16#0;
   DP_DIAG10[2] := B#16#0;
   DP_DIAG10[3] := B#16#0;
   DP_DIAG10[4] := B#16#0;
   DP_DIAG10[5] := B#16#0;
   DP_DIAG10[6] := B#16#0;
   DP_DIAG10[7] := B#16#0;
   DP_DIAG10[8] := B#16#0;
   DP_DIAG10[9] := B#16#0;
   DP_DIAG10[10] := B#16#0;
   DP_DIAG10[11] := B#16#0;
   DP_DIAG10[12] := B#16#0;
   DP_DIAG10[13] := B#16#0;
   DP_DIAG10[14] := B#16#0;
   DP_DIAG10[15] := B#16#0;
   DP_DIAG10[16] := B#16#0;
   DP_DIAG10[17] := B#16#0;
   DP_DIAG10[18] := B#16#0;
   DP_DIAG10[19] := B#16#0;
   DP_DIAG10[20] := B#16#0;
   DP_DIAG10[21] := B#16#0;
   DP_DIAG10[22] := B#16#0;
   DP_DIAG10[23] := B#16#0;
   DP_DIAG10[24] := B#16#0;
   DP_DIAG10[25] := B#16#0;
   DP_DIAG10[26] := B#16#0;
   DP_DIAG10[27] := B#16#0;
   DP_DIAG10[28] := B#16#0;
   DP_DIAG10[29] := B#16#0;
   DP_DIAG10[30] := B#16#0;
   DP_DIAG10[31] := B#16#0;
   DP_DIAG10[32] := B#16#0;
   DP_DIAG10[33] := B#16#0;
   DP_DIAG10[34] := B#16#0;
   DP_DIAG10[35] := B#16#0;
   DP_DIAG10[36] := B#16#0;
   DP_DIAG10[37] := B#16#0;
   DP_DIAG10[38] := B#16#0;
   DP_DIAG10[39] := B#16#0;
   DP_DIAG10[40] := B#16#0;
   DP_DIAG10[41] := B#16#0;
   DP_DIAG10[42] := B#16#0;
   DP_DIAG10[43] := B#16#0;
   DP_DIAG10[44] := B#16#0;
   DP_DIAG10[45] := B#16#0;
   DP_DIAG10[46] := B#16#0;
   DP_DIAG10[47] := B#16#0;
   DP_DIAG10[48] := B#16#0;
   DP_DIAG10[49] := B#16#0;
   DP_DIAG10[50] := B#16#0;
   DP_DIAG10[51] := B#16#0;
   DP_DIAG10[52] := B#16#0;
   DP_DIAG10[53] := B#16#0;
   DP_DIAG10[54] := B#16#0;
   DP_DIAG10[55] := B#16#0;
   DP_DIAG10[56] := B#16#0;
   DP_DIAG10[57] := B#16#0;
   DP_DIAG10[58] := B#16#0;
   DP_DIAG10[59] := B#16#0;
   DP_DIAG10[60] := B#16#0;
   DP_DIAG10[61] := B#16#0;
   DP_DIAG10[62] := B#16#0;
   DP_DIAG10[63] := B#16#0;
   DP_DIAG10[64] := B#16#0;
   DP_DIAG10[65] := B#16#0;
   DP_DIAG10[66] := B#16#0;
   DP_DIAG10[67] := B#16#0;
   DP_DIAG10[68] := B#16#0;
   DP_DIAG10[69] := B#16#0;
   DP_DIAG10[70] := B#16#0;
   DP_DIAG10[71] := B#16#0;
   DP_DIAG10[72] := B#16#0;
   DP_DIAG10[73] := B#16#0;
   DP_DIAG10[74] := B#16#0;
   DP_DIAG10[75] := B#16#0;
   DP_DIAG10[76] := B#16#0;
   DP_DIAG10[77] := B#16#0;
   DP_DIAG10[78] := B#16#0;
   DP_DIAG10[79] := B#16#0;
   DP_DIAG10[80] := B#16#0;
   DP_DIAG10[81] := B#16#0;
   DP_DIAG10[82] := B#16#0;
   DP_DIAG10[83] := B#16#0;
   DP_DIAG10[84] := B#16#0;
   DP_DIAG10[85] := B#16#0;
   DP_DIAG10[86] := B#16#0;
   DP_DIAG10[87] := B#16#0;
   DP_DIAG10[88] := B#16#0;
   DP_DIAG10[89] := B#16#0;
   DP_DIAG10[90] := B#16#0;
   DP_DIAG10[91] := B#16#0;
   DP_DIAG10[92] := B#16#0;
   DP_DIAG10[93] := B#16#0;
   DP_DIAG10[94] := B#16#0;
   DP_DIAG10[95] := B#16#0;
   DP_DIAG10[96] := B#16#0;
   DP_DIAG10[97] := B#16#0;
   DP_DIAG10[98] := B#16#0;
   DP_DIAG10[99] := B#16#0;
   DP_DIAG10[100] := B#16#0;
END_DATA_BLOCK

DATA_BLOCK DB 486
TITLE =Interface Data Block (PLC<==>611U)
VERSION : 0.1


  STRUCT
   Send : UDT 1000;
   Receive : UDT 2000;
   Axis_Pos : REAL ;	//Axis Current Pos
  END_STRUCT ;
BEGIN
   Send.STW1.Bit_8 := FALSE;
   Send.STW1.Bit_9 := FALSE;
   Send.STW1.Bit_10 := FALSE;
   Send.STW1.Bit_11 := FALSE;
   Send.STW1.Bit_12 := FALSE;
   Send.STW1.Bit_13 := FALSE;
   Send.STW1.Bit_14 := FALSE;
   Send.STW1.Bit_15 := FALSE;
   Send.STW1.Bit_0 := FALSE;
   Send.STW1.Bit_1 := FALSE;
   Send.STW1.Bit_2 := FALSE;
   Send.STW1.Bit_3 := FALSE;
   Send.STW1.Bit_4 := FALSE;
   Send.STW1.Bit_5 := FALSE;
   Send.STW1.Bit_6 := FALSE;
   Send.STW1.Bit_7 := FALSE;
   Send.SatzAnw.BLKSEL := 0;
   Send.PosStw.Bit_8 := FALSE;
   Send.PosStw.Bit_9 := FALSE;
   Send.PosStw.Bit_10 := FALSE;
   Send.PosStw.Bit_11 := FALSE;
   Send.PosStw.Bit_12 := FALSE;
   Send.PosStw.Bit_13 := FALSE;
   Send.PosStw.Bit_14 := FALSE;
   Send.PosStw.Bit_15 := FALSE;
   Send.PosStw.Bit_0 := FALSE;
   Send.PosStw.Bit_1 := FALSE;
   Send.PosStw.Bit_2 := FALSE;
   Send.PosStw.Bit_3 := FALSE;
   Send.PosStw.Bit_4 := FALSE;
   Send.PosStw.Bit_5 := FALSE;
   Send.PosStw.Bit_6 := FALSE;
   Send.PosStw.Bit_7 := FALSE;
   Send.STW2.Bit_8 := FALSE;
   Send.STW2.Bit_9 := FALSE;
   Send.STW2.Bit_10 := FALSE;
   Send.STW2.Bit_11 := FALSE;
   Send.STW2.Bit_12 := FALSE;
   Send.STW2.Bit_13 := FALSE;
   Send.STW2.Bit_14 := FALSE;
   Send.STW2.Bit_15 := FALSE;
   Send.STW2.Bit_0 := FALSE;
   Send.STW2.Bit_1 := FALSE;
   Send.STW2.Bit_2 := FALSE;
   Send.STW2.Bit_3 := FALSE;
   Send.STW2.Bit_4 := FALSE;
   Send.STW2.Bit_5 := FALSE;
   Send.STW2.Bit_6 := FALSE;
   Send.STW2.Bit_7 := FALSE;
   Send.Over.Override := 0;
   Send.Temp1 := 0;
   Send.Temp2 := 0;
   Send.Temp3 := 0;
   Send.Temp4 := 0;
   Send.Temp5 := 0;
   Receive.ZSW1.Bit_8 := FALSE;
   Receive.ZSW1.Bit_9 := FALSE;
   Receive.ZSW1.Bit_10 := FALSE;
   Receive.ZSW1.Bit_11 := FALSE;
   Receive.ZSW1.Bit_12 := FALSE;
   Receive.ZSW1.Bir_13 := FALSE;
   Receive.ZSW1.Bit_14 := FALSE;
   Receive.ZSW1.Bit_15 := FALSE;
   Receive.ZSW1.Bit_0 := FALSE;
   Receive.ZSW1.Bit_1 := FALSE;
   Receive.ZSW1.Bit_2 := FALSE;
   Receive.ZSW1.Bit_3 := FALSE;
   Receive.ZSW1.Bit_4 := FALSE;
   Receive.ZSW1.Bit_5 := FALSE;
   Receive.ZSW1.Bit_6 := FALSE;
   Receive.ZSW1.Bit_7 := FALSE;
   Receive.AktSatz.CURRBLK := 1024;
   Receive.PosZsw.Bit_8 := FALSE;
   Receive.PosZsw.Bit_9 := FALSE;
   Receive.PosZsw.Bit_10 := FALSE;
   Receive.PosZsw.Bit_11 := FALSE;
   Receive.PosZsw.Bit_12 := FALSE;
   Receive.PosZsw.Bit_13 := FALSE;
   Receive.PosZsw.Bit_14 := FALSE;
   Receive.PosZsw.Bit_15 := FALSE;
   Receive.PosZsw.Bit_0 := FALSE;
   Receive.PosZsw.Bit_1 := FALSE;
   Receive.PosZsw.Bit_2 := FALSE;
   Receive.PosZsw.Bit_3 := FALSE;
   Receive.PosZsw.Bit_4 := FALSE;
   Receive.PosZsw.Bit_5 := FALSE;
   Receive.PosZsw.Bit_6 := FALSE;
   Receive.PosZsw.Bit_7 := FALSE;
   Receive.ZSW2.Bit_8 := FALSE;
   Receive.ZSW2.Bit_9 := FALSE;
   Receive.ZSW2.Bit_10 := FALSE;
   Receive.ZSW2.Bit_11 := FALSE;
   Receive.ZSW2.Bit_12 := FALSE;
   Receive.ZSW2.Bit_13 := FALSE;
   Receive.ZSW2.Bit_14 := FALSE;
   Receive.ZSW2.Bit_15 := FALSE;
   Receive.ZSW2.Bit_0 := FALSE;
   Receive.ZSW2.Bit_1 := FALSE;
   Receive.ZSW2.Bit_2 := FALSE;
   Receive.ZSW2.Bit_3 := FALSE;
   Receive.ZSW2.Bit_4 := FALSE;
   Receive.ZSW2.Bit_5 := FALSE;
   Receive.ZSW2.Bit_6 := FALSE;
   Receive.ZSW2.Bit_7 := FALSE;
   Receive.MessW.Bit_8 := FALSE;
   Receive.MessW.Bit_9 := FALSE;
   Receive.MessW.Bit_10 := FALSE;
   Receive.MessW.Bit_11 := FALSE;
   Receive.MessW.Bit_12 := FALSE;
   Receive.MessW.Bit_13 := FALSE;
   Receive.MessW.Bit_14 := FALSE;
   Receive.MessW.Bit_15 := FALSE;
   Receive.MessW.Bit_0 := FALSE;
   Receive.MessW.Bit_1 := FALSE;
   Receive.MessW.Bit_2 := FALSE;
   Receive.MessW.Bit_3 := FALSE;
   Receive.MessW.Bit_4 := FALSE;
   Receive.MessW.Bit_5 := FALSE;
   Receive.MessW.Bit_6 := FALSE;
   Receive.MessW.Bit_7 := FALSE;
   Receive.XactP1 := W#16#0;
   Receive.XactP2 := W#16#0;
   Receive.Temp1 := 0;
   Receive.Temp2 := 0;
   Receive.Temp3 := 0;
   Axis_Pos := 1.310690e+002;
END_DATA_BLOCK

FUNCTION FC 486 : VOID
TITLE =Simodrive 611U Control Function
//P102 : 모터 최대 이송속도
//P103 : 최대가속
//P104 : 최대감속
//
//P108 : 수동이송1 속도
//P109 : 수동이송2 속도
//
//P200:8 => Kv factor (Position Control Gain)
//
//P314 : 소프트 리미트 활성화
//P315 : 마이너스 소프트 리미트 값
//P316 : 플러스 소프트 리미트 값
//
//P700 : 제어모드
//       0 : 드라이브 사용안함 (드라이브 B만사용시)
//       1 : 스피트/토르크 제어
//       2 : 위치셋 포인트 제어
//       3 : 위치제어
//
//주의: P1012.12를 0으로 만들것. Power on Inihnbit
//P1012 = 4104h 로 설정
//
//Profibus Parameterization --> Frame Selection ==> 0으로 설정 (사용자화)
VERSION : 0.1


VAR_INPUT
  Enable : BOOL ;	//Always On or Ready
  Jog_Cw : BOOL ;	//수동 축이송 + 신호
  Jog_Ccw : BOOL ;	//수동 축이송 - 신호
  Target_Pos : INT ;	//자동 이송 목표위치 번호
  Start : BOOL ;	//자동 목표위치 이동 시작
  Override_10 : BOOL ;	//저속신호
  Override_100 : BOOL ;	//고속신호
  Em_Stop : BOOL ;	//비상정지 신호 (정상시 신호 On 되어있음, NC)
  Reset : BOOL ;	//리셋신호
END_VAR
VAR_OUTPUT
  Ref_Reach : BOOL ;	//축 원점복귀 완료신호
  Fault : BOOL ;	//Simodrive 611U 이상
  Pos_Reach : BOOL ;	//목표위치 도달신호
  Current_Pos : REAL ;	//축 현재위치
END_VAR
VAR_TEMP
  Send_Ret : INT ;
  Receive_Ret : INT ;
END_VAR
BEGIN
NETWORK
TITLE =Process Data Send (PLC==>611U)
//PZD Start Address = 264
//LADDR = W#16#108 ==> DEC 264
//PPO5 이므로, 전체를 사용하지 않더라도 20Byte 를 전송한다.
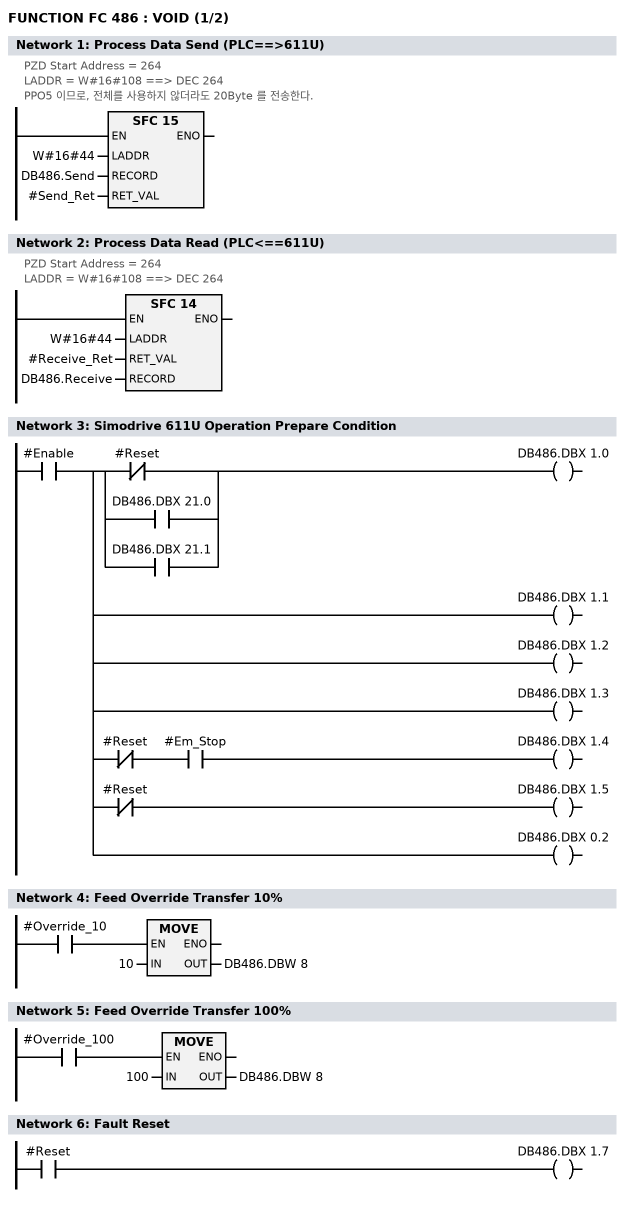
      CALL SFC   15 (
           LADDR                    := W#16#44,
           RECORD                   := DB486.Send,
           RET_VAL                  := #Send_Ret);
      NOP   0;
NETWORK
TITLE =Process Data Read (PLC<==611U)
//PZD Start Address = 264
//LADDR = W#16#108 ==> DEC 264
      CALL SFC   14 (
           LADDR                    := W#16#44,
           RET_VAL                  := #Receive_Ret,
           RECORD                   := DB486.Receive);
      NOP   0;
NETWORK
TITLE =Simodrive 611U Operation Prepare Condition
//
//
      A     #Enable;
      =     L      4.0;
      A     L      4.0;
      A(    ;
      ON    #Reset;
      O     DB486.DBX   21.0;
      O     DB486.DBX   21.1;
      )     ;
      =     DB486.DBX    1.0;
      A     L      4.0;
      BLD   102;
      =     DB486.DBX    1.1;
      A     L      4.0;
      BLD   102;
      =     DB486.DBX    1.2;
      A     L      4.0;
      BLD   102;
      =     DB486.DBX    1.3;
      A     L      4.0;
      AN    #Reset;
      A     #Em_Stop;
      =     DB486.DBX    1.4;
      A     L      4.0;
      AN    #Reset;
      =     DB486.DBX    1.5;
      A     L      4.0;
      BLD   102;
      =     DB486.DBX    0.2;
NETWORK
TITLE =Feed Override Transfer 10%

      A     #Override_10;
      JNB   _001;
      L     10;
      T     DB486.DBW    8;
_001: NOP   0;
NETWORK
TITLE =Feed Override Transfer 100%

      A     #Override_100;
      JNB   _002;
      L     100;
      T     DB486.DBW    8;
_002: NOP   0;
NETWORK
TITLE =Fault Reset

      A     #Reset;
      =     DB486.DBX    1.7;
NETWORK
TITLE =Jog Move 1 (Plus Direction)
//Parameter 108 ==> Fixed Setpoint
//조그이송1과 조그이송2가 동시에 on 되면, 에러가 발생됨 주의
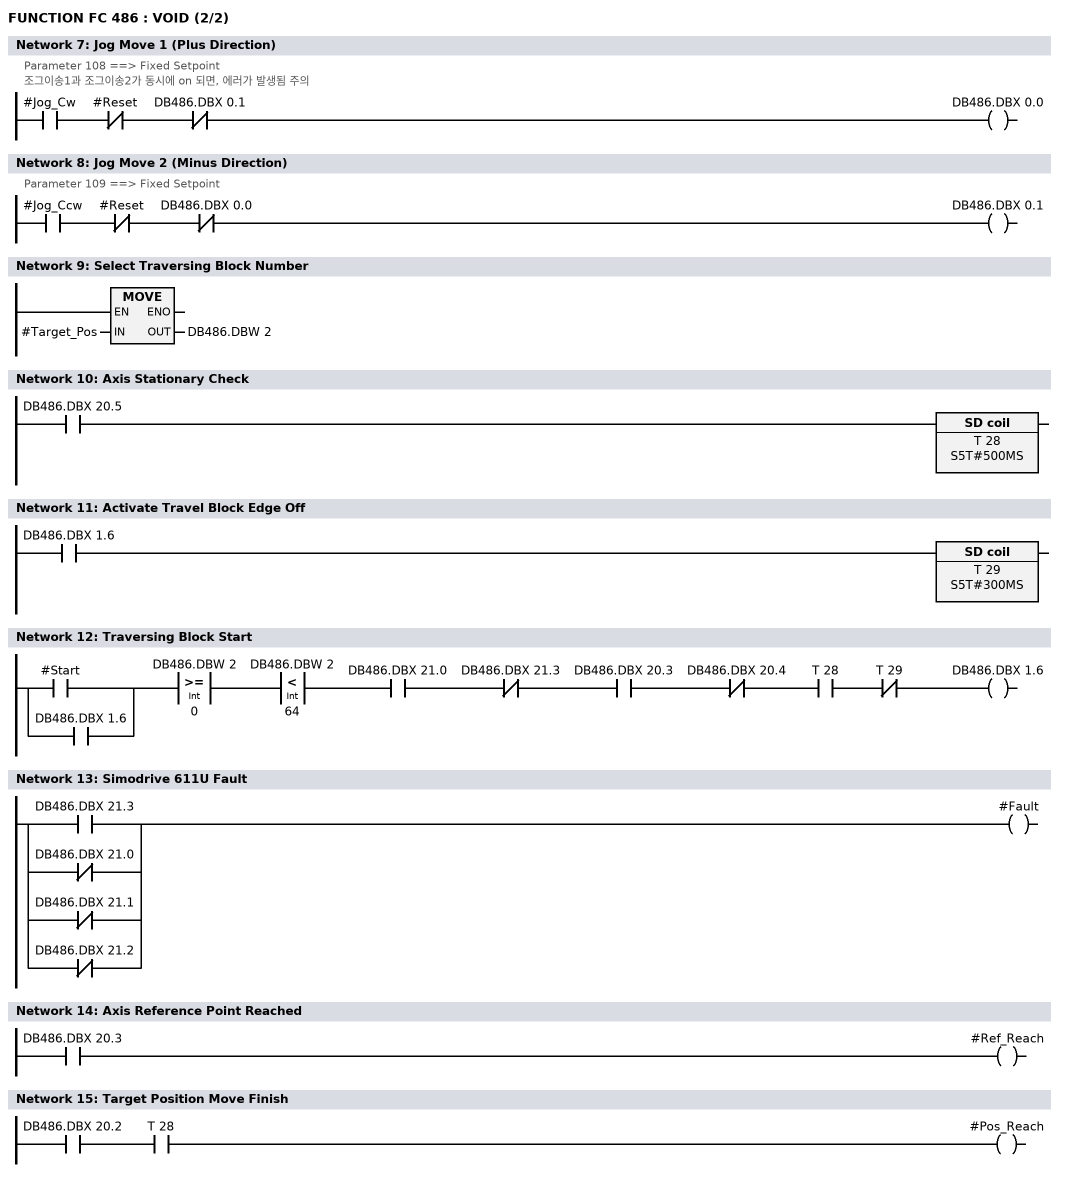
      A     #Jog_Cw;
      AN    #Reset;
      AN    DB486.DBX    0.1;
      =     DB486.DBX    0.0;
NETWORK
TITLE =Jog Move 2 (Minus Direction)
//Parameter 109 ==> Fixed Setpoint
      A     #Jog_Ccw;
      AN    #Reset;
      AN    DB486.DBX    0.0;
      =     DB486.DBX    0.1;
NETWORK
TITLE =Select Traversing Block Number

      L     #Target_Pos;
      T     DB486.DBW    2;
      NOP   0;
NETWORK
TITLE =Axis Stationary Check

      A     DB486.DBX   20.5;
      L     S5T#500MS;
      SD    T     28;
NETWORK
TITLE =Activate Travel Block Edge Off

      A     DB486.DBX    1.6;
      L     S5T#300MS;
      SD    T     29;
NETWORK
TITLE =Traversing Block Start

      A(    ;
      O     #Start;
      O     DB486.DBX    1.6;
      )     ;
      A(    ;
      L     DB486.DBW    2;
      L     0;
      >=I   ;
      )     ;
      A(    ;
      L     DB486.DBW    2;
      L     64;
      <I    ;
      )     ;
      A     DB486.DBX   21.0;
      AN    DB486.DBX   21.3;
      A     DB486.DBX   20.3;
      AN    DB486.DBX   20.4;
      A     T     28;
      AN    T     29;
      =     DB486.DBX    1.6;
NETWORK
TITLE =Simodrive 611U Fault

      O     DB486.DBX   21.3;
      ON    DB486.DBX   21.0;
      ON    DB486.DBX   21.1;
      ON    DB486.DBX   21.2;
      =     #Fault;
NETWORK
TITLE =Axis Reference Point Reached

      A     DB486.DBX   20.3;
      =     #Ref_Reach;
NETWORK
TITLE =Target Position Move Finish

      A     DB486.DBX   20.2;
      A     T     28;
      =     #Pos_Reach;
NETWORK
TITLE =Axis Current Pos Calculate

      L     DB486.DBD   30;
      DTR   ;
      T     DB486.DBD   40;

      L     DB486.DBD   40;
      L     1.000000e+003; // db120.dbd40/1000.0
      /R    ;
      T     DB486.DBD   40;
      T     #Current_Pos;


NETWORK
TITLE =Reference Point Start
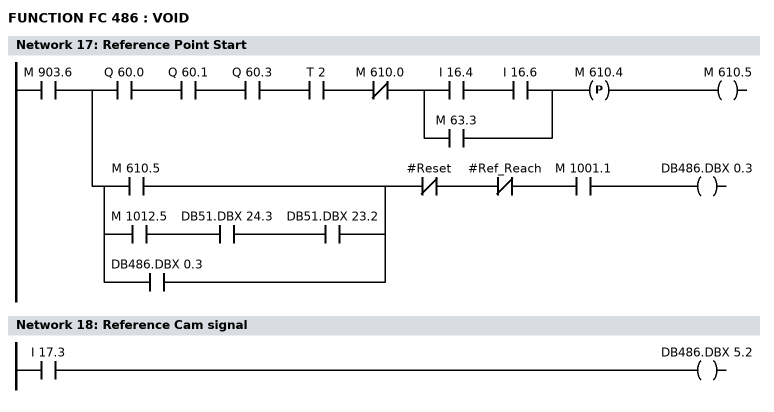

      A     M    903.6;
      =     L      4.0;
      A     L      4.0;
      A     Q     60.0;
      A     Q     60.1;
      A     Q     60.3;
      A     T      2;
      AN    M    610.0;
      A(    ;
      A     I     16.4;
      A     I     16.6;
      O     M     63.3;
      )     ;
      FP    M    610.4;
      =     M    610.5;
      A     L      4.0;
      A(    ;
      O     M    610.5;
      O     ;
      A     M   1012.5;
      A     DB51.DBX   24.3;
      A     DB51.DBX   23.2;
      O     DB486.DBX    0.3;
      )     ;
      AN    #Reset;
      AN    #Ref_Reach;
      A     M   1001.1;
      =     DB486.DBX    0.3;
NETWORK
TITLE =Reference Cam signal

      A     I     17.3;
      =     DB486.DBX    5.2;
END_FUNCTION

FUNCTION FC 98 : VOID
TITLE =
VERSION : 0.1


VAR_TEMP
  SFC20_RET_VAL : INT ;
  RECV1_LEN : WORD ;
  SEND1_LEN : WORD ;
  RECV2_LEN : WORD ;
  SEND2_LEN : WORD ;
END_VAR
BEGIN
NETWORK
TITLE =
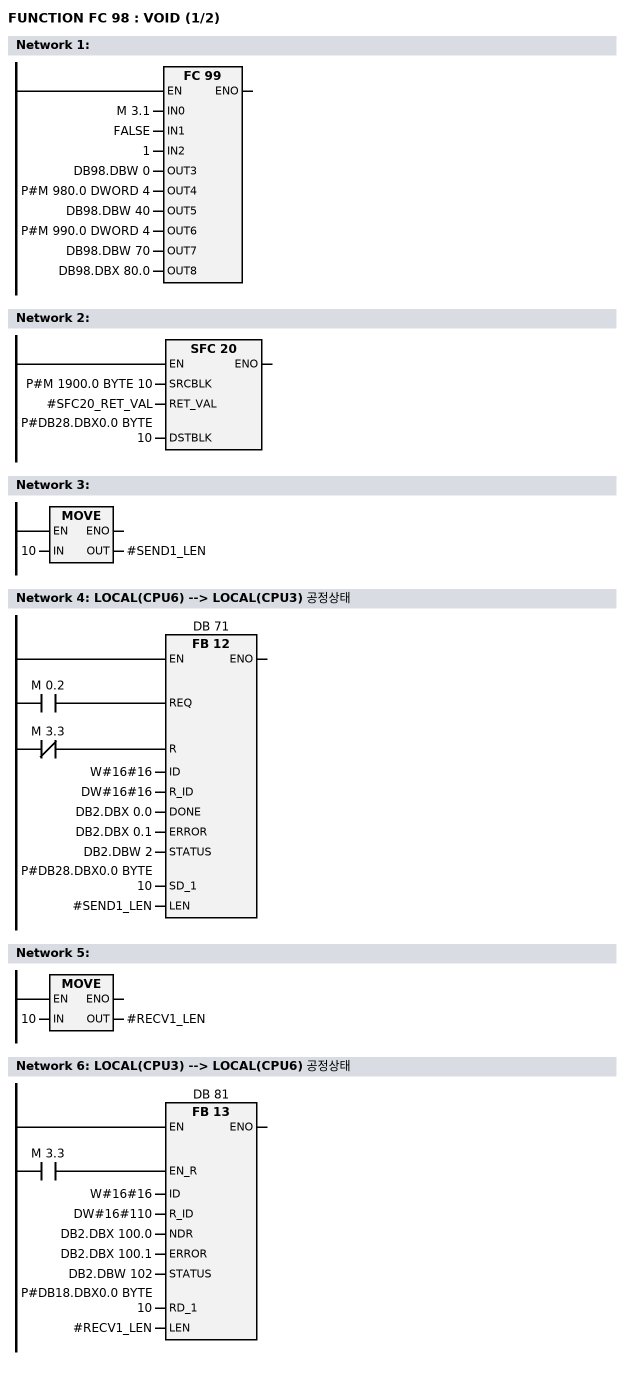

      CALL FC    99 (
           IN0                      := M      3.1,
           IN1                      := FALSE,
           IN2                      := 1,
           OUT3                     := DB98.DBW    0,
           OUT4                     := P#M 980.0 DWORD 4,
           OUT5                     := DB98.DBW   40,
           OUT6                     := P#M 990.0 DWORD 4,
           OUT7                     := DB98.DBW   70,
           OUT8                     := DB98.DBX   80.0);
NETWORK
TITLE =

      CALL SFC   20 (
           SRCBLK                   := P#M 1900.0 BYTE 10,
           RET_VAL                  := #SFC20_RET_VAL,
           DSTBLK                   := P#DB28.DBX0.0 BYTE 10);
      NOP   0;
NETWORK
TITLE =

      L     10;
      T     #SEND1_LEN;
      NOP   0;
NETWORK
TITLE =LOCAL(CPU6) --> LOCAL(CPU3) 공정상태

      A     M      0.2;
      =     L     10.0;
      BLD   103;
      AN    M      3.3;
      =     L     10.1;
      BLD   103;
      CALL FB    12 , DB    71 (
           REQ                      := L     10.0,
           R                        := L     10.1,
           ID                       := W#16#16,
           R_ID                     := DW#16#16,
           DONE                     := DB2.DBX    0.0,
           ERROR                    := DB2.DBX    0.1,
           STATUS                   := DB2.DBW    2,
           SD_1                     := P#DB28.DBX0.0 BYTE 10,
           LEN                      := #SEND1_LEN);
      NOP   0;
NETWORK
TITLE =

      L     10;
      T     #RECV1_LEN;
      NOP   0;
NETWORK
TITLE =LOCAL(CPU3) --> LOCAL(CPU6) 공정상태

      A     M      3.3;
      =     L     10.0;
      BLD   103;
      CALL FB    13 , DB    81 (
           EN_R                     := L     10.0,
           ID                       := W#16#16,
           R_ID                     := DW#16#110,
           NDR                      := DB2.DBX  100.0,
           ERROR                    := DB2.DBX  100.1,
           STATUS                   := DB2.DBW  102,
           RD_1                     := P#DB18.DBX0.0 BYTE 10,
           LEN                      := #RECV1_LEN);
      NOP   0;
NETWORK
TITLE =
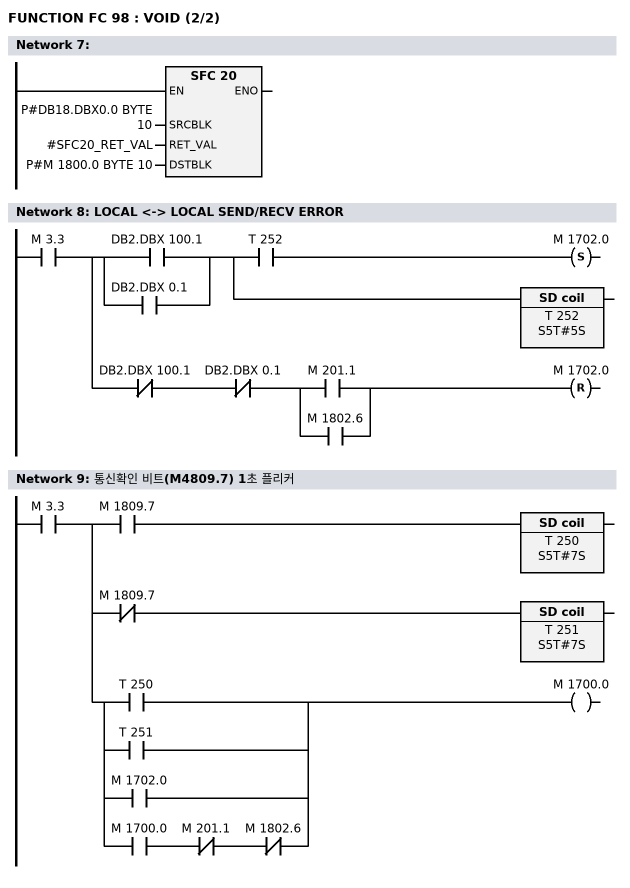

      CALL SFC   20 (
           SRCBLK                   := P#DB18.DBX0.0 BYTE 10,
           RET_VAL                  := #SFC20_RET_VAL,
           DSTBLK                   := P#M 1800.0 BYTE 10);
      NOP   0;
NETWORK
TITLE =LOCAL <-> LOCAL SEND/RECV ERROR

      A     M      3.3;
      =     L     10.0;
      A     L     10.0;
      A(    ;
      O     DB2.DBX  100.1;
      O     DB2.DBX    0.1;
      )     ;
      =     L     10.1;
      A     L     10.1;
      A     T    252;
      S     M   1702.0;
      A     L     10.1;
      BLD   102;
      L     S5T#5S;
      SD    T    252;
      A     L     10.0;
      AN    DB2.DBX  100.1;
      AN    DB2.DBX    0.1;
      A(    ;
      O     M    201.1;
      O     M   1802.6;
      )     ;
      R     M   1702.0;
NETWORK
TITLE =통신확인 비트(M4809.7) 1초 플리커
//
//
//
      A     M      3.3;
      =     L     10.0;
      A     L     10.0;
      A     M   1809.7;
      L     S5T#7S;
      SD    T    250;
      A     L     10.0;
      AN    M   1809.7;
      L     S5T#7S;
      SD    T    251;
      A     L     10.0;
      A(    ;
      O     T    250;
      O     T    251;
      O     M   1702.0;
      O     ;
      A     M   1700.0;
      AN    M    201.1;
      AN    M   1802.6;
      )     ;
      =     M   1700.0;
END_FUNCTION

FUNCTION FC 114 : VOID
TITLE =
VERSION : 0.1

BEGIN
NETWORK
TITLE =
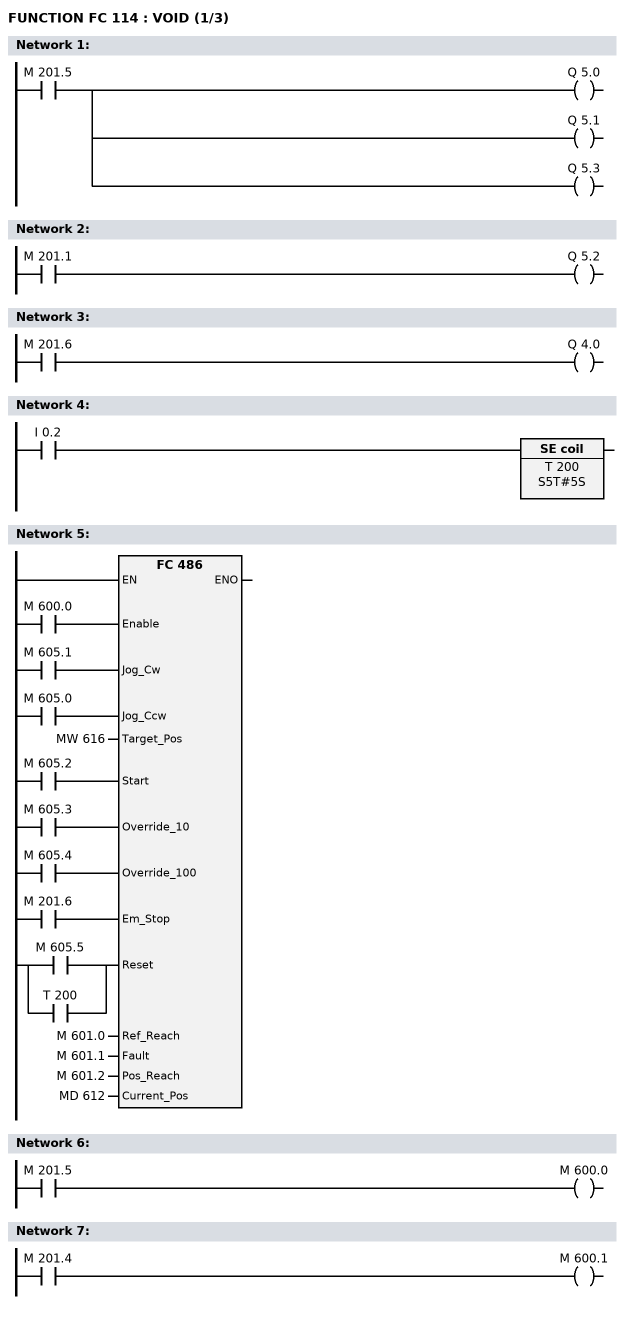

      A     M    201.5;
      =     Q      5.0;
      =     Q      5.1;
      =     Q      5.3;
NETWORK
TITLE =

      A     M    201.1;
      =     Q      5.2;
NETWORK
TITLE =

      A     M    201.6;
      =     Q      4.0;
NETWORK
TITLE =

      A     I      0.2;
      L     S5T#5S;
      SE    T    200;
NETWORK
TITLE =

      A     M    600.0;
      =     L      0.0;
      BLD   103;
      A     M    605.1;
      =     L      0.1;
      BLD   103;
      A     M    605.0;
      =     L      0.2;
      BLD   103;
      A     M    605.2;
      =     L      0.3;
      BLD   103;
      A     M    605.3;
      =     L      0.4;
      BLD   103;
      A     M    605.4;
      =     L      0.5;
      BLD   103;
      A     M    201.6;
      =     L      0.6;
      BLD   103;
      A(    ;
      O     M    605.5;
      O     T    200;
      )     ;
      =     L      0.7;
      BLD   103;
      CALL FC   486 (
           Enable                   := L      0.0,
           Jog_Cw                   := L      0.1,
           Jog_Ccw                  := L      0.2,
           Target_Pos               := MW   616,
           Start                    := L      0.3,
           Override_10              := L      0.4,
           Override_100             := L      0.5,
           Em_Stop                  := L      0.6,
           Reset                    := L      0.7,
           Ref_Reach                := M    601.0,
           Fault                    := M    601.1,
           Pos_Reach                := M    601.2,
           Current_Pos              := MD   612);
      NOP   0;
NETWORK
TITLE =

      A     M    201.5;
      =     M    600.0;
NETWORK
TITLE =

      A     M    201.4;
      =     M    600.1;
NETWORK
TITLE =
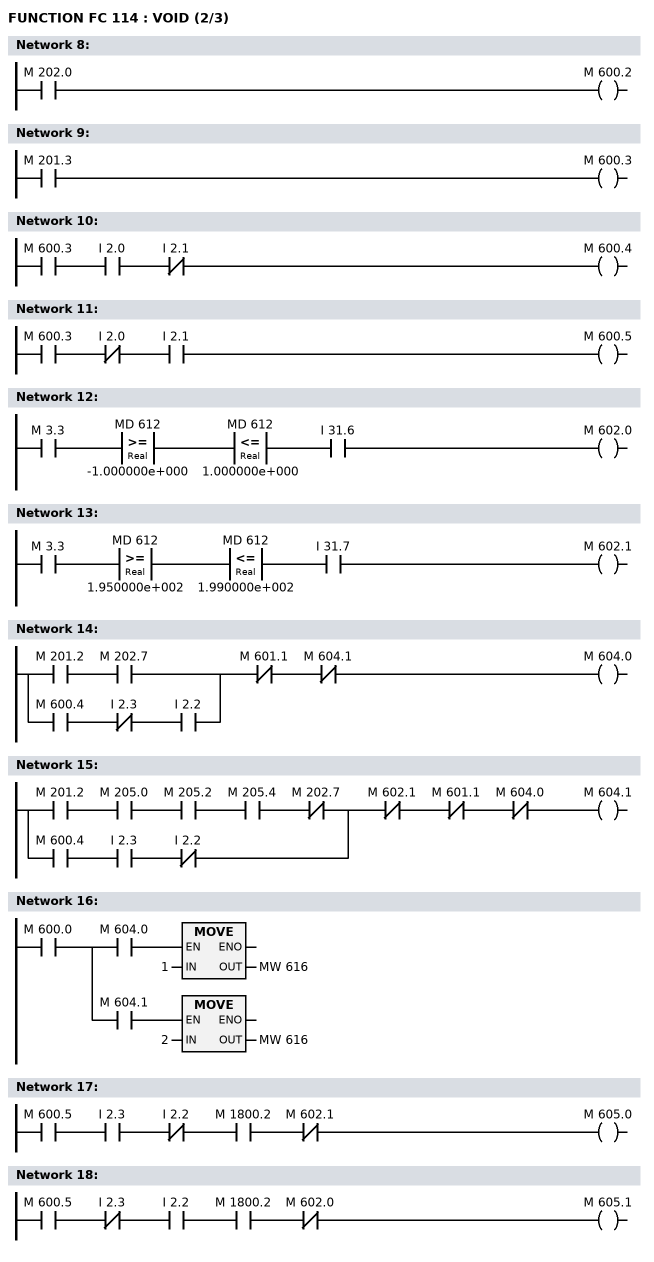

      A     M    202.0;
      =     M    600.2;
NETWORK
TITLE =

      A     M    201.3;
      =     M    600.3;
NETWORK
TITLE =

      A     M    600.3;
      A     I      2.0;
      AN    I      2.1;
      =     M    600.4;
NETWORK
TITLE =

      A     M    600.3;
      AN    I      2.0;
      A     I      2.1;
      =     M    600.5;
NETWORK
TITLE =

      A     M      3.3;
      A(    ;
      L     MD   612;
      L     -1.000000e+000;
      >=R   ;
      )     ;
      A(    ;
      L     MD   612;
      L     1.000000e+000;
      <=R   ;
      )     ;
      A     I     31.6;
      =     M    602.0;
NETWORK
TITLE =

      A     M      3.3;
      A(    ;
      L     MD   612;
      L     1.950000e+002;
      >=R   ;
      )     ;
      A(    ;
      L     MD   612;
      L     1.990000e+002;
      <=R   ;
      )     ;
      A     I     31.7;
      =     M    602.1;
NETWORK
TITLE =

      A(    ;
      A     M    201.2;
      A     M    202.7;
      O     ;
      A     M    600.4;
      AN    I      2.3;
      A     I      2.2;
      )     ;
      AN    M    601.1;
      AN    M    604.1;
      =     M    604.0;
NETWORK
TITLE =

      A(    ;
      A     M    201.2;
      A     M    205.0;
      A     M    205.2;
      A     M    205.4;
      AN    M    202.7;
      O     ;
      A     M    600.4;
      A     I      2.3;
      AN    I      2.2;
      )     ;
      AN    M    602.1;
      AN    M    601.1;
      AN    M    604.0;
      =     M    604.1;
NETWORK
TITLE =

      A     M    600.0;
      =     L      0.0;
      A     L      0.0;
      A     M    604.0;
      JNB   _001;
      L     1;
      T     MW   616;
_001: NOP   0;
      A     L      0.0;
      A     M    604.1;
      JNB   _002;
      L     2;
      T     MW   616;
_002: NOP   0;
NETWORK
TITLE =

      A     M    600.5;
      A     I      2.3;
      AN    I      2.2;
      A     M   1800.2;
      AN    M    602.1;
      =     M    605.0;
NETWORK
TITLE =

      A     M    600.5;
      AN    I      2.3;
      A     I      2.2;
      A     M   1800.2;
      AN    M    602.0;
      =     M    605.1;
NETWORK
TITLE =
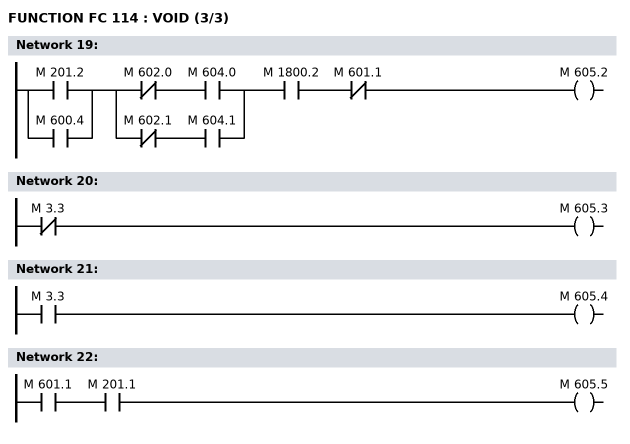

      A(    ;
      O     M    201.2;
      O     M    600.4;
      )     ;
      A(    ;
      AN    M    602.0;
      A     M    604.0;
      O     ;
      AN    M    602.1;
      A     M    604.1;
      )     ;
      A     M   1800.2;
      AN    M    601.1;
      =     M    605.2;
NETWORK
TITLE =

      AN    M      3.3;
      =     M    605.3;
NETWORK
TITLE =

      A     M      3.3;
      =     M    605.4;
NETWORK
TITLE =

      A     M    601.1;
      A     M    201.1;
      =     M    605.5;
END_FUNCTION

FUNCTION FC 130 : VOID
TITLE =
VERSION : 0.1

BEGIN
NETWORK
TITLE =
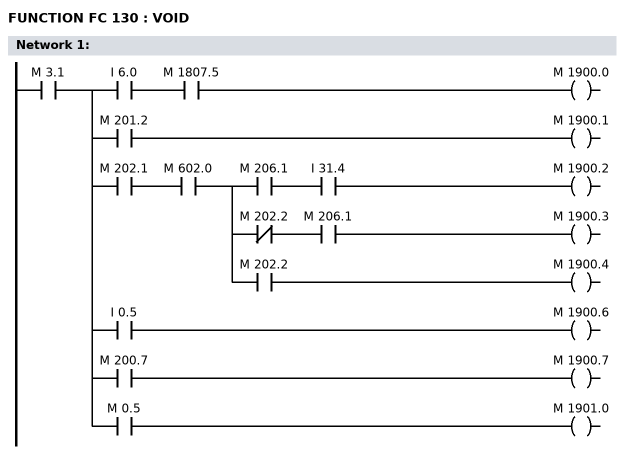

      A     M      3.1;
      =     L      0.0;
      A     L      0.0;
      A     I      6.0;
      A     M   1807.5;
      =     M   1900.0;
      A     L      0.0;
      A     M    201.2;
      =     M   1900.1;
      A     L      0.0;
      A     M    202.1;
      A     M    602.0;
      =     L      0.1;
      A     L      0.1;
      A     M    206.1;
      A     I     31.4;
      =     M   1900.2;
      A     L      0.1;
      AN    M    202.2;
      A     M    206.1;
      =     M   1900.3;
      A     L      0.1;
      A     M    202.2;
      =     M   1900.4;
      A     L      0.0;
      A     I      0.5;
      =     M   1900.6;
      A     L      0.0;
      A     M    200.7;
      =     M   1900.7;
      A     L      0.0;
      A     M      0.5;
      =     M   1901.0;
END_FUNCTION

FUNCTION FC 200 : VOID
TITLE =
VERSION : 0.1

BEGIN
NETWORK
TITLE =
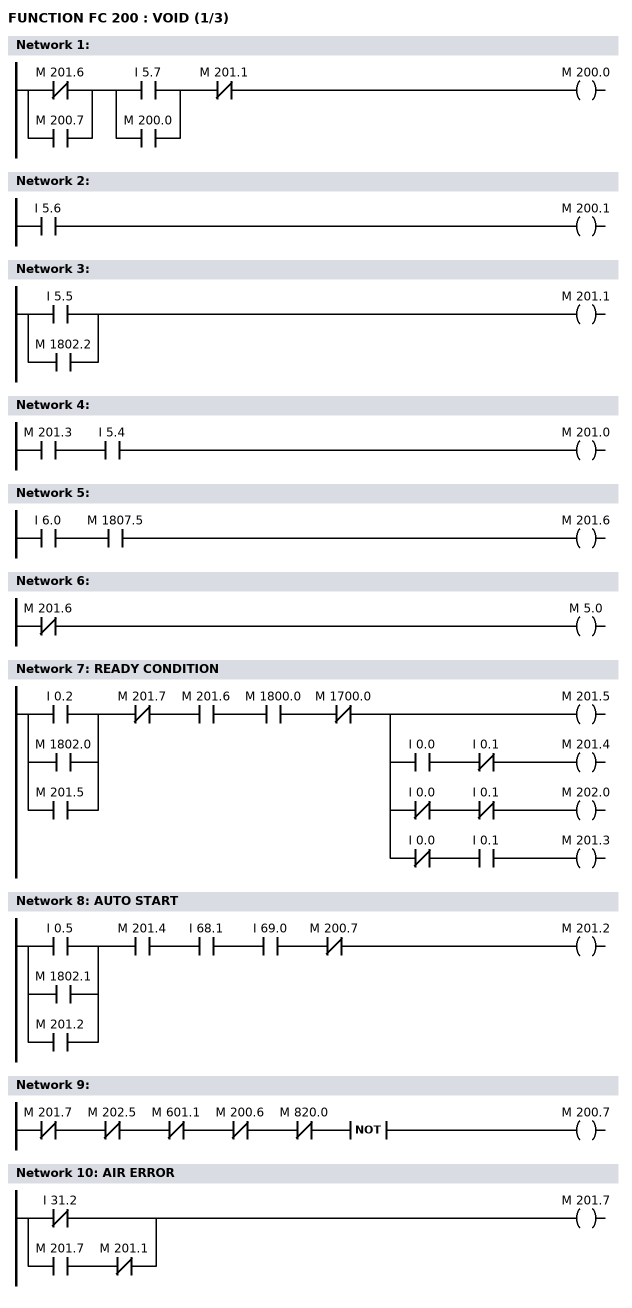

      A(    ;
      ON    M    201.6;
      O     M    200.7;
      )     ;
      A(    ;
      O     I      5.7;
      O     M    200.0;
      )     ;
      AN    M    201.1;
      =     M    200.0;
NETWORK
TITLE =

      A     I      5.6;
      =     M    200.1;
NETWORK
TITLE =

      O     I      5.5;
      O     M   1802.2;
      =     M    201.1;
NETWORK
TITLE =

      A     M    201.3;
      A     I      5.4;
      =     M    201.0;
NETWORK
TITLE =

      A     I      6.0;
      A     M   1807.5;
      =     M    201.6;
NETWORK
TITLE =

      AN    M    201.6;
      =     M      5.0;
NETWORK
TITLE =READY CONDITION

